LIN {X 0.018,Y -426.505,Z 505.911,A 0.000,B 0.000,C 90.000,E1 199.939} C_DIS
LIN {X 0.001,Y -422.220,Z 505.894,A 0.000,B 0.000,C 90.000,E1 196.913} C_DIS
LIN {X 0.056,Y -419.219,Z 505.881,A 0.000,B 0.000,C 90.000,E1 194.537} C_DIS
LIN {X -0.079,Y -416.405,Z 505.868,A 0.000,B 0.000,C 90.000,E1 192.175} C_DIS
LIN {X -0.186,Y -414.138,Z 505.856,A 0.000,B 0.000,C 90.000,E1 190.141} C_DIS
LIN {X 0.071,Y -411.990,Z 505.845,A 0.000,B 0.000,C 90.000,E1 188.049} C_DIS
LIN {X 0.180,Y -410.282,Z 505.835,A 0.000,B 0.000,C 90.000,E1 186.315} C_DIS
LIN {X 0.176,Y -407.524,Z 505.820,A 0.000,B 0.000,C 90.000,E1 183.555} C_DIS
LIN {X 0.039,Y -405.409,Z 505.805,A 0.000,B 0.000,C 90.000,E1 180.802} C_DIS
LIN {X -0.121,Y -404.165,Z 505.793,A 0.000,B 0.000,C 90.000,E1 178.740} C_DIS
LIN {X -0.033,Y -402.565,Z 505.770,A 0.000,B 0.000,C 90.000,E1 174.546} C_DIS
LIN {X 0.172,Y -402.279,Z 505.752,A 0.000,B 0.000,C 90.000,E1 171.376} C_DIS
LIN {X 0.214,Y -402.491,Z 505.739,A 0.000,B 0.000,C 90.000,E1 168.926} C_DIS
LIN {X -0.118,Y -402.858,Z 505.729,A 0.000,B 0.000,C 90.000,E1 167.229} C_DIS
LIN {X 0.210,Y -403.708,Z 505.714,A 0.000,B 0.000,C 90.000,E1 164.393} C_DIS
LIN {X 0.006,Y -405.079,Z 505.698,A 0.000,B 0.000,C 90.000,E1 161.638} C_DIS
LIN {X -0.119,Y -406.382,Z 505.686,A 0.000,B 0.000,C 90.000,E1 159.571} C_DIS
LIN {X 0.038,Y -409.257,Z 505.665,A 0.000,B 0.000,C 90.000,E1 155.741} C_DIS
LIN {X -0.103,Y -411.046,Z 505.654,A 0.000,B 0.000,C 90.000,E1 153.691} C_DIS
LIN {X -0.125,Y -412.516,Z 505.644,A 0.000,B 0.000,C 90.000,E1 151.975} C_DIS
LIN {X -0.098,Y -413.912,Z 505.635,A 0.000,B 0.000,C 90.000,E1 150.255} C_DIS
LIN {X -0.039,Y -415.256,Z 505.625,A 0.000,B 0.000,C 90.000,E1 148.535} C_DIS
LIN {X -0.093,Y -416.520,Z 505.616,A 0.000,B 0.000,C 90.000,E1 146.834} C_DIS
LIN {X 0.055,Y -417.849,Z 505.604,A 0.000,B 0.000,C 90.000,E1 144.769} C_DIS
LIN {X 0.184,Y -418.995,Z 505.595,A 0.000,B 0.000,C 90.000,E1 143.050} C_DIS
LIN {X 0.008,Y -420.032,Z 505.585,A 0.000,B 0.000,C 90.000,E1 141.376} C_DIS
LIN {X 0.116,Y -420.969,Z 505.576,A 0.000,B 0.000,C 90.000,E1 139.666} C_DIS
LIN {X 0.124,Y -421.898,Z 505.565,A 0.000,B 0.000,C 90.000,E1 137.634} C_DIS
LIN {X 0.116,Y -422.218,Z 505.559,A 0.000,B 0.000,C 90.000,E1 136.620} C_DIS
LIN {X 0.203,Y -422.557,Z 505.550,A 0.000,B 0.000,C 90.000,E1 134.919} C_DIS
LIN {X -0.099,Y -422.626,Z 505.544,A 0.000,B 0.000,C 90.000,E1 133.947} C_DIS
LIN {X -0.198,Y -422.402,Z 505.537,A 0.000,B 0.000,C 90.000,E1 132.609} C_DIS
LIN {X -0.199,Y -421.973,Z 505.531,A 0.000,B 0.000,C 90.000,E1 131.595} C_DIS
LIN {X -0.003,Y -421.086,Z 505.523,A 0.000,B 0.000,C 90.000,E1 130.216} C_DIS
LIN {X 0.024,Y -420.265,Z 505.518,A 0.000,B 0.000,C 90.000,E1 129.197} C_DIS
LIN {X -0.139,Y -418.800,Z 505.508,A 0.000,B 0.000,C 90.000,E1 127.523} C_DIS
LIN {X 0.000,Y -417.194,Z 505.499,A 0.000,B 0.000,C 90.000,E1 125.804} C_DIS
LIN {X -0.124,Y -416.814,Z 505.497,A 0.000,B 0.000,C 90.000,E1 125.438} C_DIS
LIN {X -0.161,Y -416.824,Z 505.497,A 0.000,B 0.000,C 90.000,E1 125.438} C_DIS
LIN {X 0.103,Y -426.391,Z 505.476,A 0.000,B 0.000,C 90.000,E1 121.720} C_DIS
LIN {X 0.058,Y -430.444,Z 505.469,A 0.000,B 0.000,C 90.000,E1 120.384} C_DIS
LIN {X -0.155,Y -432.036,Z 505.465,A 0.000,B 0.000,C 90.000,E1 119.745} C_DIS
LIN {X -0.164,Y -441.367,Z 505.445,A 0.000,B 0.000,C 90.000,E1 116.104} C_DIS
LIN {X 0.152,Y -444.273,Z 505.439,A 0.000,B 0.000,C 90.000,E1 115.079} C_DIS
LIN {X 0.005,Y -445.126,Z 505.438,A 0.000,B 0.000,C 90.000,E1 114.771} C_DIS
LIN {X 0.113,Y -454.300,Z 505.416,A 0.000,B 0.000,C 90.000,E1 110.865} C_DIS
LIN {X -0.196,Y -456.967,Z 505.411,A 0.000,B 0.000,C 90.000,E1 109.939} C_DIS
LIN {X 0.042,Y -458.234,Z 505.407,A 0.000,B 0.000,C 90.000,E1 109.268} C_DIS
LIN {X 0.191,Y -460.170,Z 505.401,A 0.000,B 0.000,C 90.000,E1 108.236} C_DIS
LIN {X 0.164,Y -460.188,Z 505.401,A 0.000,B 0.000,C 90.000,E1 108.236} C_DIS
LIN {X -0.031,Y -477.013,Z 505.399,A 0.000,B 0.000,C 90.000,E1 107.819} C_DIS
LIN {X 0.118,Y -487.752,Z 505.397,A 0.000,B 0.000,C 90.000,E1 107.511} C_DIS
LIN {X 0.183,Y -501.865,Z 505.395,A 0.000,B 0.000,C 90.000,E1 107.094} C_DIS
LIN {X -0.084,Y -512.281,Z 505.393,A 0.000,B 0.000,C 90.000,E1 106.804} C_DIS
LIN {X 0.104,Y -522.750,Z 505.391,A 0.000,B 0.000,C 90.000,E1 106.441} C_DIS
LIN {X 0.115,Y -533.203,Z 505.389,A 0.000,B 0.000,C 90.000,E1 106.079} C_DIS
LIN {X -0.021,Y -539.788,Z 505.388,A 0.000,B 0.000,C 90.000,E1 105.843} C_DIS
LIN {X 0.026,Y -549.515,Z 505.386,A 0.000,B 0.000,C 90.000,E1 105.426} C_DIS
LIN {X -0.055,Y -556.133,Z 505.384,A 0.000,B 0.000,C 90.000,E1 105.134} C_DIS
LIN {X -0.214,Y -562.178,Z 505.382,A 0.000,B 0.000,C 90.000,E1 104.828} C_DIS
LIN {X 0.204,Y -568.361,Z 505.380,A 0.000,B 0.000,C 90.000,E1 104.426} C_DIS
LIN {X -0.021,Y -574.397,Z 505.378,A 0.000,B 0.000,C 90.000,E1 104.064} C_DIS
LIN {X 0.015,Y -580.246,Z 505.376,A 0.000,B 0.000,C 90.000,E1 103.647} C_DIS
LIN {X -0.165,Y -585.770,Z 505.373,A 0.000,B 0.000,C 90.000,E1 103.231} C_DIS
LIN {X -0.180,Y -591.131,Z 505.371,A 0.000,B 0.000,C 90.000,E1 102.771} C_DIS
LIN {X -0.036,Y -598.036,Z 505.367,A 0.000,B 0.000,C 90.000,E1 102.119} C_DIS
LIN {X -0.101,Y -605.453,Z 505.363,A 0.000,B 0.000,C 90.000,E1 101.366} C_DIS
LIN {X -0.084,Y -609.662,Z 505.361,A 0.000,B 0.000,C 90.000,E1 100.894} C_DIS
LIN {X -0.103,Y -613.896,Z 505.358,A 0.000,B 0.000,C 90.000,E1 100.423} C_DIS
LIN {X 0.123,Y -618.926,Z 505.355,A 0.000,B 0.000,C 90.000,E1 99.792} C_DIS
LIN {X 0.104,Y -623.916,Z 505.351,A 0.000,B 0.000,C 90.000,E1 99.151} C_DIS
LIN {X -0.027,Y -629.277,Z 505.347,A 0.000,B 0.000,C 90.000,E1 98.398} C_DIS
LIN {X -0.108,Y -634.217,Z 505.342,A 0.000,B 0.000,C 90.000,E1 97.644} C_DIS
LIN {X -0.145,Y -638.618,Z 505.338,A 0.000,B 0.000,C 90.000,E1 96.891} C_DIS
LIN {X -0.088,Y -641.983,Z 505.335,A 0.000,B 0.000,C 90.000,E1 96.258} C_DIS
LIN {X 0.000,Y -645.065,Z 505.331,A 0.000,B 0.000,C 90.000,E1 95.625} C_DIS
LIN {X -0.178,Y -649.744,Z 505.326,A 0.000,B 0.000,C 90.000,E1 94.645} C_DIS
LIN {X -0.141,Y -652.900,Z 505.322,A 0.000,B 0.000,C 90.000,E1 93.898} C_DIS
LIN {X 0.094,Y -654.803,Z 505.319,A 0.000,B 0.000,C 90.000,E1 93.383} C_DIS
LIN {X -0.274,Y -656.487,Z 505.316,A 0.000,B 0.000,C 90.000,E1 92.922} C_DIS
LIN {X -0.010,Y -657.988,Z 505.313,A 0.000,B 0.000,C 90.000,E1 92.407} C_DIS
LIN {X 0.105,Y -659.741,Z 505.309,A 0.000,B 0.000,C 90.000,E1 91.661} C_DIS
LIN {X -0.264,Y -660.700,Z 505.307,A 0.000,B 0.000,C 90.000,E1 91.203} C_DIS
LIN {X 0.037,Y -661.322,Z 505.304,A 0.000,B 0.000,C 90.000,E1 90.688} C_DIS
LIN {X -0.319,Y -661.735,Z 505.301,A 0.000,B 0.000,C 90.000,E1 90.229} C_DIS
LIN {X -0.009,Y -661.834,Z 505.298,A 0.000,B 0.000,C 90.000,E1 89.714} C_DIS
LIN {X 0.126,Y -661.721,Z 505.294,A 0.000,B 0.000,C 90.000,E1 88.969} C_DIS
LIN {X 0.255,Y -661.045,Z 505.290,A 0.000,B 0.000,C 90.000,E1 88.224} C_DIS
LIN {X -0.080,Y -660.385,Z 505.288,A 0.000,B 0.000,C 90.000,E1 87.764} C_DIS
LIN {X 0.032,Y -658.956,Z 505.284,A 0.000,B 0.000,C 90.000,E1 87.020} C_DIS
LIN {X -0.305,Y -657.826,Z 505.281,A 0.000,B 0.000,C 90.000,E1 86.560} C_DIS
LIN {X -0.032,Y -656.465,Z 505.278,A 0.000,B 0.000,C 90.000,E1 86.045} C_DIS
LIN {X 0.275,Y -654.873,Z 505.275,A 0.000,B 0.000,C 90.000,E1 85.527} C_DIS
LIN {X -0.287,Y -652.156,Z 505.271,A 0.000,B 0.000,C 90.000,E1 84.837} C_DIS
LIN {X -0.004,Y -650.150,Z 505.268,A 0.000,B 0.000,C 90.000,E1 84.318} C_DIS
LIN {X 0.036,Y -646.773,Z 505.264,A 0.000,B 0.000,C 90.000,E1 83.571} C_DIS
LIN {X 0.279,Y -644.240,Z 505.262,A 0.000,B 0.000,C 90.000,E1 83.053} C_DIS
LIN {X -0.180,Y -640.958,Z 505.258,A 0.000,B 0.000,C 90.000,E1 82.470} C_DIS
LIN {X -0.058,Y -636.731,Z 505.254,A 0.000,B 0.000,C 90.000,E1 81.724} C_DIS
LIN {X -0.022,Y -630.363,Z 505.249,A 0.000,B 0.000,C 90.000,E1 80.735} C_DIS
LIN {X -0.110,Y -624.978,Z 505.244,A 0.000,B 0.000,C 90.000,E1 79.982} C_DIS
LIN {X 0.086,Y -619.367,Z 505.240,A 0.000,B 0.000,C 90.000,E1 79.218} C_DIS
LIN {X 0.134,Y -614.176,Z 505.237,A 0.000,B 0.000,C 90.000,E1 78.578} C_DIS
LIN {X 0.062,Y -608.507,Z 505.233,A 0.000,B 0.000,C 90.000,E1 77.937} C_DIS
LIN {X 0.169,Y -603.608,Z 505.230,A 0.000,B 0.000,C 90.000,E1 77.409} C_DIS
LIN {X -0.064,Y -598.510,Z 505.227,A 0.000,B 0.000,C 90.000,E1 76.937} C_DIS
LIN {X -0.120,Y -593.055,Z 505.225,A 0.000,B 0.000,C 90.000,E1 76.464} C_DIS
LIN {X 0.014,Y -587.480,Z 505.222,A 0.000,B 0.000,C 90.000,E1 75.992} C_DIS
LIN {X 0.273,Y -581.520,Z 505.220,A 0.000,B 0.000,C 90.000,E1 75.519} C_DIS
LIN {X -0.186,Y -575.580,Z 505.218,A 0.000,B 0.000,C 90.000,E1 75.172} C_DIS
LIN {X -0.012,Y -570.706,Z 505.216,A 0.000,B 0.000,C 90.000,E1 74.866} C_DIS
LIN {X -0.110,Y -563.793,Z 505.214,A 0.000,B 0.000,C 90.000,E1 74.519} C_DIS
LIN {X -0.172,Y -558.480,Z 505.213,A 0.000,B 0.000,C 90.000,E1 74.283} C_DIS
LIN {X 0.162,Y -553.060,Z 505.211,A 0.000,B 0.000,C 90.000,E1 74.031} C_DIS
LIN {X 0.016,Y -545.580,Z 505.210,A 0.000,B 0.000,C 90.000,E1 73.795} C_DIS
LIN {X 0.160,Y -539.833,Z 505.209,A 0.000,B 0.000,C 90.000,E1 73.614} C_DIS
LIN {X 0.030,Y -532.141,Z 505.208,A 0.000,B 0.000,C 90.000,E1 73.449} C_DIS
LIN {X -0.123,Y -523.817,Z 505.207,A 0.000,B 0.000,C 90.000,E1 73.323} C_DIS
LIN {X -0.043,Y -511.657,Z 505.206,A 0.000,B 0.000,C 90.000,E1 73.142} C_DIS
LIN {X 0.061,Y -500.841,Z 505.206,A 0.000,B 0.000,C 90.000,E1 73.015} C_DIS
LIN {X 0.175,Y -495.888,Z 505.206,A 0.000,B 0.000,C 90.000,E1 72.960} C_DIS
LIN {X -0.166,Y -488.331,Z 505.205,A 0.000,B 0.000,C 90.000,E1 72.960} C_DIS
LIN {X 0.119,Y -478.178,Z 505.205,A 0.000,B 0.000,C 90.000,E1 72.851} C_DIS
LIN {X -0.010,Y -474.985,Z 505.205,A 0.000,B 0.000,C 90.000,E1 72.851} C_DIS
LIN {X -0.042,Y -474.946,Z 505.205,A 0.000,B 0.000,C 90.000,E1 72.851} C_DIS
LIN {X 0.221,Y -474.159,Z 505.201,A 0.000,B 0.000,C 90.000,E1 72.054} C_DIS
LIN {X 0.088,Y -465.644,Z 505.173,A 0.000,B 0.000,C 90.000,E1 67.050} C_DIS
LIN {X -0.033,Y -456.637,Z 505.148,A 0.000,B 0.000,C 90.000,E1 62.615} C_DIS
LIN {X -0.034,Y -455.594,Z 505.144,A 0.000,B 0.000,C 90.000,E1 61.975} C_DIS
LIN {X 0.150,Y -452.503,Z 505.137,A 0.000,B 0.000,C 90.000,E1 60.667} C_DIS
LIN {X -0.182,Y -448.840,Z 505.128,A 0.000,B 0.000,C 90.000,E1 59.076} C_DIS
LIN {X -0.221,Y -448.858,Z 505.128,A 0.000,B 0.000,C 90.000,E1 59.076} C_DIS
LIN {X 0.196,Y -453.401,Z 505.122,A 0.000,B 0.000,C 90.000,E1 57.916} C_DIS
LIN {X 0.110,Y -457.127,Z 505.117,A 0.000,B 0.000,C 90.000,E1 56.962} C_DIS
LIN {X -0.044,Y -458.885,Z 505.114,A 0.000,B 0.000,C 90.000,E1 56.501} C_DIS
LIN {X -0.200,Y -461.027,Z 505.110,A 0.000,B 0.000,C 90.000,E1 55.881} C_DIS
LIN {X 0.048,Y -463.771,Z 505.105,A 0.000,B 0.000,C 90.000,E1 54.895} C_DIS
LIN {X -0.072,Y -465.454,Z 505.102,A 0.000,B 0.000,C 90.000,E1 54.276} C_DIS
LIN {X -0.145,Y -467.569,Z 505.096,A 0.000,B 0.000,C 90.000,E1 53.336} C_DIS
LIN {X 0.042,Y -468.814,Z 505.093,A 0.000,B 0.000,C 90.000,E1 52.683} C_DIS
LIN {X 0.013,Y -470.423,Z 505.088,A 0.000,B 0.000,C 90.000,E1 51.743} C_DIS
LIN {X -0.148,Y -472.508,Z 505.079,A 0.000,B 0.000,C 90.000,E1 50.194} C_DIS
LIN {X -0.059,Y -473.786,Z 505.072,A 0.000,B 0.000,C 90.000,E1 48.933} C_DIS
LIN {X -0.093,Y -474.575,Z 505.067,A 0.000,B 0.000,C 90.000,E1 48.000} C_DIS
LIN {X -0.115,Y -475.209,Z 505.061,A 0.000,B 0.000,C 90.000,E1 47.067} C_DIS
LIN {X -0.132,Y -475.735,Z 505.056,A 0.000,B 0.000,C 90.000,E1 46.134} C_DIS
LIN {X 0.187,Y -476.122,Z 505.051,A 0.000,B 0.000,C 90.000,E1 45.162} C_DIS
LIN {X -0.055,Y -476.457,Z 505.044,A 0.000,B 0.000,C 90.000,E1 43.947} C_DIS
LIN {X 0.050,Y -476.486,Z 505.037,A 0.000,B 0.000,C 90.000,E1 42.690} C_DIS
LIN {X 0.152,Y -476.221,Z 505.030,A 0.000,B 0.000,C 90.000,E1 41.434} C_DIS
LIN {X -0.171,Y -475.911,Z 505.025,A 0.000,B 0.000,C 90.000,E1 40.539} C_DIS
LIN {X 0.059,Y -475.261,Z 505.017,A 0.000,B 0.000,C 90.000,E1 38.955} C_DIS
LIN {X 0.133,Y -474.287,Z 505.006,A 0.000,B 0.000,C 90.000,E1 37.076} C_DIS
LIN {X -0.098,Y -473.158,Z 504.996,A 0.000,B 0.000,C 90.000,E1 35.231} C_DIS
LIN {X -0.016,Y -472.070,Z 504.987,A 0.000,B 0.000,C 90.000,E1 33.658} C_DIS
LIN {X -0.011,Y -470.371,Z 504.975,A 0.000,B 0.000,C 90.000,E1 31.465} C_DIS
LIN {X -0.075,Y -468.725,Z 504.964,A 0.000,B 0.000,C 90.000,E1 29.589} C_DIS
LIN {X -0.226,Y -467.068,Z 504.954,A 0.000,B 0.000,C 90.000,E1 27.719} C_DIS
LIN {X 0.012,Y -465.525,Z 504.943,A 0.000,B 0.000,C 90.000,E1 25.796} C_DIS
LIN {X 0.013,Y -464.076,Z 504.933,A 0.000,B 0.000,C 90.000,E1 23.898} C_DIS
LIN {X -0.143,Y -463.094,Z 504.924,A 0.000,B 0.000,C 90.000,E1 22.333} C_DIS
LIN {X -0.138,Y -462.053,Z 504.913,A 0.000,B 0.000,C 90.000,E1 20.429} C_DIS
LIN {X 0.122,Y -461.156,Z 504.903,A 0.000,B 0.000,C 90.000,E1 18.489} C_DIS
LIN {X -0.090,Y -460.199,Z 504.889,A 0.000,B 0.000,C 90.000,E1 15.969} C_DIS
LIN {X -0.025,Y -459.576,Z 504.875,A 0.000,B 0.000,C 90.000,E1 13.411} C_DIS
LIN {X -0.068,Y -459.439,Z 504.859,A 0.000,B 0.000,C 90.000,E1 10.546} C_DIS
LIN {X 0.229,Y -459.695,Z 504.846,A 0.000,B 0.000,C 90.000,E1 8.276} C_DIS
LIN {X -0.113,Y -460.288,Z 504.834,A 0.000,B 0.000,C 90.000,E1 6.087} C_DIS
LIN {X 0.026,Y -461.345,Z 504.821,A 0.000,B 0.000,C 90.000,E1 3.841} C_DIS
LIN {X -0.104,Y -462.522,Z 504.811,A 0.000,B 0.000,C 90.000,E1 1.949} C_DIS
LIN {X 0.000,Y -463.977,Z 504.800,A 0.000,B 0.000,C 90.000,E1 360.000} C_DIS
LIN {X -0.123,Y -466.352,Z 504.787,A 0.000,B 0.000,C 90.000,E1 357.593} C_DIS
LIN {X -0.128,Y -467.758,Z 504.780,A 0.000,B 0.000,C 90.000,E1 356.331} C_DIS
LIN {X -0.046,Y -470.034,Z 504.769,A 0.000,B 0.000,C 90.000,E1 354.432} C_DIS
LIN {X 0.038,Y -471.673,Z 504.762,A 0.000,B 0.000,C 90.000,E1 353.166} C_DIS
LIN {X 0.028,Y -473.689,Z 504.753,A 0.000,B 0.000,C 90.000,E1 351.602} C_DIS
LIN {X -0.109,Y -477.718,Z 504.738,A 0.000,B 0.000,C 90.000,E1 348.814} C_DIS
LIN {X 0.182,Y -482.461,Z 504.722,A 0.000,B 0.000,C 90.000,E1 345.992} C_DIS
LIN {X -0.059,Y -486.669,Z 504.710,A 0.000,B 0.000,C 90.000,E1 343.866} C_DIS
LIN {X 0.069,Y -491.080,Z 504.698,A 0.000,B 0.000,C 90.000,E1 341.710} C_DIS
LIN {X 0.038,Y -493.709,Z 504.692,A 0.000,B 0.000,C 90.000,E1 340.496} C_DIS
LIN {X 0.219,Y -496.330,Z 504.685,A 0.000,B 0.000,C 90.000,E1 339.263} C_DIS
LIN {X -0.198,Y -498.964,Z 504.678,A 0.000,B 0.000,C 90.000,E1 338.103} C_DIS
LIN {X 0.135,Y -502.099,Z 504.670,A 0.000,B 0.000,C 90.000,E1 336.561} C_DIS
LIN {X 0.186,Y -504.564,Z 504.663,A 0.000,B 0.000,C 90.000,E1 335.357} C_DIS
LIN {X -0.003,Y -508.099,Z 504.653,A 0.000,B 0.000,C 90.000,E1 333.589} C_DIS
LIN {X -0.108,Y -511.728,Z 504.643,A 0.000,B 0.000,C 90.000,E1 331.820} C_DIS
LIN {X -0.117,Y -515.345,Z 504.634,A 0.000,B 0.000,C 90.000,E1 330.049} C_DIS
LIN {X 0.281,Y -518.532,Z 504.625,A 0.000,B 0.000,C 90.000,E1 328.535} C_DIS
LIN {X 0.174,Y -522.910,Z 504.614,A 0.000,B 0.000,C 90.000,E1 326.501} C_DIS
LIN {X 0.029,Y -527.428,Z 504.603,A 0.000,B 0.000,C 90.000,E1 324.482} C_DIS
LIN {X -0.106,Y -531.268,Z 504.593,A 0.000,B 0.000,C 90.000,E1 322.763} C_DIS
LIN {X -0.159,Y -534.444,Z 504.585,A 0.000,B 0.000,C 90.000,E1 321.331} C_DIS
LIN {X -0.241,Y -537.576,Z 504.577,A 0.000,B 0.000,C 90.000,E1 319.908} C_DIS
LIN {X 0.103,Y -541.341,Z 504.568,A 0.000,B 0.000,C 90.000,E1 318.162} C_DIS
LIN {X 0.124,Y -545.103,Z 504.558,A 0.000,B 0.000,C 90.000,E1 316.458} C_DIS
LIN {X 0.209,Y -548.704,Z 504.549,A 0.000,B 0.000,C 90.000,E1 314.757} C_DIS
LIN {X -0.052,Y -551.588,Z 504.541,A 0.000,B 0.000,C 90.000,E1 313.380} C_DIS
LIN {X 0.190,Y -555.091,Z 504.532,A 0.000,B 0.000,C 90.000,E1 311.676} C_DIS
LIN {X 0.062,Y -558.036,Z 504.524,A 0.000,B 0.000,C 90.000,E1 310.297} C_DIS
LIN {X 0.148,Y -561.549,Z 504.515,A 0.000,B 0.000,C 90.000,E1 308.624} C_DIS
LIN {X -0.022,Y -565.611,Z 504.504,A 0.000,B 0.000,C 90.000,E1 306.710} C_DIS
LIN {X -0.326,Y -569.663,Z 504.493,A 0.000,B 0.000,C 90.000,E1 304.818} C_DIS
LIN {X -0.191,Y -573.145,Z 504.484,A 0.000,B 0.000,C 90.000,E1 303.166} C_DIS
LIN {X -0.128,Y -575.988,Z 504.477,A 0.000,B 0.000,C 90.000,E1 301.799} C_DIS
LIN {X -0.169,Y -578.181,Z 504.471,A 0.000,B 0.000,C 90.000,E1 300.718} C_DIS
LIN {X 0.173,Y -580.786,Z 504.463,A 0.000,B 0.000,C 90.000,E1 299.333} C_DIS
LIN {X -0.231,Y -583.361,Z 504.456,A 0.000,B 0.000,C 90.000,E1 298.025} C_DIS
LIN {X -0.080,Y -585.405,Z 504.448,A 0.000,B 0.000,C 90.000,E1 296.668} C_DIS
LIN {X -0.156,Y -587.042,Z 504.441,A 0.000,B 0.000,C 90.000,E1 295.335} C_DIS
LIN {X 0.026,Y -587.805,Z 504.436,A 0.000,B 0.000,C 90.000,E1 294.515} C_DIS
LIN {X 0.176,Y -588.749,Z 504.427,A 0.000,B 0.000,C 90.000,E1 292.898} C_DIS
LIN {X 0.014,Y -589.864,Z 504.417,A 0.000,B 0.000,C 90.000,E1 291.046} C_DIS
LIN {X -0.012,Y -590.652,Z 504.408,A 0.000,B 0.000,C 90.000,E1 289.450} C_DIS
LIN {X 0.216,Y -590.968,Z 504.402,A 0.000,B 0.000,C 90.000,E1 288.362} C_DIS
LIN {X 0.136,Y -591.213,Z 504.395,A 0.000,B 0.000,C 90.000,E1 287.040} C_DIS
LIN {X 0.200,Y -591.371,Z 504.389,A 0.000,B 0.000,C 90.000,E1 285.969} C_DIS
LIN {X -0.036,Y -591.454,Z 504.382,A 0.000,B 0.000,C 90.000,E1 284.662} C_DIS
LIN {X -0.010,Y -591.469,Z 504.373,A 0.000,B 0.000,C 90.000,E1 283.063} C_DIS
LIN {X 0.145,Y -591.396,Z 504.362,A 0.000,B 0.000,C 90.000,E1 281.186} C_DIS
LIN {X -0.092,Y -591.179,Z 504.353,A 0.000,B 0.000,C 90.000,E1 279.613} C_DIS
LIN {X -0.023,Y -590.906,Z 504.346,A 0.000,B 0.000,C 90.000,E1 278.276} C_DIS
LIN {X 0.138,Y -590.415,Z 504.337,A 0.000,B 0.000,C 90.000,E1 276.663} C_DIS
LIN {X -0.146,Y -589.943,Z 504.331,A 0.000,B 0.000,C 90.000,E1 275.625} C_DIS
LIN {X -0.008,Y -588.999,Z 504.322,A 0.000,B 0.000,C 90.000,E1 274.012} C_DIS
LIN {X -0.172,Y -587.921,Z 504.315,A 0.000,B 0.000,C 90.000,E1 272.694} C_DIS
LIN {X 0.236,Y -586.563,Z 504.307,A 0.000,B 0.000,C 90.000,E1 271.318} C_DIS
LIN {X -0.171,Y -585.335,Z 504.302,A 0.000,B 0.000,C 90.000,E1 270.286} C_DIS
LIN {X -0.224,Y -583.438,Z 504.293,A 0.000,B 0.000,C 90.000,E1 268.682} C_DIS
LIN {X 0.273,Y -581.327,Z 504.284,A 0.000,B 0.000,C 90.000,E1 267.020} C_DIS
LIN {X 0.015,Y -579.543,Z 504.276,A 0.000,B 0.000,C 90.000,E1 265.698} C_DIS
LIN {X -0.266,Y -577.635,Z 504.269,A 0.000,B 0.000,C 90.000,E1 264.375} C_DIS
LIN {X 0.185,Y -575.024,Z 504.260,A 0.000,B 0.000,C 90.000,E1 262.704} C_DIS
LIN {X 0.079,Y -572.312,Z 504.251,A 0.000,B 0.000,C 90.000,E1 261.084} C_DIS
LIN {X 0.008,Y -569.624,Z 504.241,A 0.000,B 0.000,C 90.000,E1 259.454} C_DIS
LIN {X -0.186,Y -567.135,Z 504.234,A 0.000,B 0.000,C 90.000,E1 258.105} C_DIS
LIN {X -0.038,Y -565.167,Z 504.228,A 0.000,B 0.000,C 90.000,E1 256.992} C_DIS
LIN {X 0.075,Y -563.100,Z 504.222,A 0.000,B 0.000,C 90.000,E1 255.880} C_DIS
LIN {X -0.108,Y -560.304,Z 504.214,A 0.000,B 0.000,C 90.000,E1 254.519} C_DIS
LIN {X -0.186,Y -557.330,Z 504.206,A 0.000,B 0.000,C 90.000,E1 253.142} C_DIS
LIN {X -0.035,Y -553.406,Z 504.197,A 0.000,B 0.000,C 90.000,E1 251.456} C_DIS
LIN {X 0.098,Y -551.385,Z 504.192,A 0.000,B 0.000,C 90.000,E1 250.604} C_DIS
LIN {X 0.033,Y -547.744,Z 504.185,A 0.000,B 0.000,C 90.000,E1 249.209} C_DIS
LIN {X 0.091,Y -544.010,Z 504.177,A 0.000,B 0.000,C 90.000,E1 247.794} C_DIS
LIN {X 0.287,Y -540.067,Z 504.169,A 0.000,B 0.000,C 90.000,E1 246.357} C_DIS
LIN {X 0.196,Y -536.721,Z 504.163,A 0.000,B 0.000,C 90.000,E1 245.229} C_DIS
LIN {X 0.195,Y -531.571,Z 504.153,A 0.000,B 0.000,C 90.000,E1 243.512} C_DIS
LIN {X -0.147,Y -526.240,Z 504.143,A 0.000,B 0.000,C 90.000,E1 241.820} C_DIS
LIN {X -0.209,Y -519.944,Z 504.132,A 0.000,B 0.000,C 90.000,E1 239.793} C_DIS
LIN {X -0.197,Y -515.403,Z 504.124,A 0.000,B 0.000,C 90.000,E1 238.329} C_DIS
LIN {X -0.002,Y -510.726,Z 504.116,A 0.000,B 0.000,C 90.000,E1 236.834} C_DIS
LIN {X -0.007,Y -504.940,Z 504.106,A 0.000,B 0.000,C 90.000,E1 235.055} C_DIS
LIN {X 0.029,Y -499.215,Z 504.096,A 0.000,B 0.000,C 90.000,E1 233.256} C_DIS
LIN {X -0.195,Y -492.849,Z 504.084,A 0.000,B 0.000,C 90.000,E1 231.170} C_DIS
LIN {X 0.194,Y -487.664,Z 504.074,A 0.000,B 0.000,C 90.000,E1 229.299} C_DIS
LIN {X 0.227,Y -481.919,Z 504.062,A 0.000,B 0.000,C 90.000,E1 227.148} C_DIS
LIN {X -0.029,Y -476.996,Z 504.052,A 0.000,B 0.000,C 90.000,E1 225.324} C_DIS
LIN {X 0.030,Y -471.503,Z 504.040,A 0.000,B 0.000,C 90.000,E1 223.137} C_DIS
LIN {X -0.007,Y -466.207,Z 504.027,A 0.000,B 0.000,C 90.000,E1 220.943} C_DIS
LIN {X -0.177,Y -461.262,Z 504.015,A 0.000,B 0.000,C 90.000,E1 218.749} C_DIS
LIN {X 0.206,Y -457.145,Z 504.005,A 0.000,B 0.000,C 90.000,E1 216.790} C_DIS
LIN {X 0.046,Y -452.546,Z 503.992,A 0.000,B 0.000,C 90.000,E1 214.565} C_DIS
LIN {X -0.157,Y -447.570,Z 503.978,A 0.000,B 0.000,C 90.000,E1 212.005} C_DIS
LIN {X -0.128,Y -443.975,Z 503.967,A 0.000,B 0.000,C 90.000,E1 210.050} C_DIS
LIN {X 0.229,Y -439.275,Z 503.952,A 0.000,B 0.000,C 90.000,E1 207.385} C_DIS
LIN {X -0.192,Y -435.760,Z 503.941,A 0.000,B 0.000,C 90.000,E1 205.463} C_DIS
LIN {X -0.087,Y -432.341,Z 503.930,A 0.000,B 0.000,C 90.000,E1 203.462} C_DIS
LIN {X -0.065,Y -429.010,Z 503.919,A 0.000,B 0.000,C 90.000,E1 201.461} C_DIS
LIN {X 0.160,Y -426.426,Z 503.910,A 0.000,B 0.000,C 90.000,E1 199.758} C_DIS
LIN {X -0.044,Y -422.596,Z 503.895,A 0.000,B 0.000,C 90.000,E1 197.094} C_DIS
LIN {X 0.024,Y -419.551,Z 503.882,A 0.000,B 0.000,C 90.000,E1 194.717} C_DIS
LIN {X -0.098,Y -416.705,Z 503.869,A 0.000,B 0.000,C 90.000,E1 192.355} C_DIS
LIN {X -0.072,Y -414.060,Z 503.855,A 0.000,B 0.000,C 90.000,E1 189.962} C_DIS
LIN {X 0.174,Y -411.896,Z 503.844,A 0.000,B 0.000,C 90.000,E1 187.871} C_DIS
LIN {X -0.179,Y -410.198,Z 503.834,A 0.000,B 0.000,C 90.000,E1 186.201} C_DIS
LIN {X -0.170,Y -408.124,Z 503.823,A 0.000,B 0.000,C 90.000,E1 184.131} C_DIS
LIN {X 0.115,Y -405.631,Z 503.806,A 0.000,B 0.000,C 90.000,E1 180.974} C_DIS
LIN {X -0.038,Y -404.364,Z 503.794,A 0.000,B 0.000,C 90.000,E1 178.912} C_DIS
LIN {X 0.023,Y -402.698,Z 503.771,A 0.000,B 0.000,C 90.000,E1 174.723} C_DIS
LIN {X -0.116,Y -402.362,Z 503.755,A 0.000,B 0.000,C 90.000,E1 171.951} C_DIS
LIN {X -0.137,Y -402.522,Z 503.742,A 0.000,B 0.000,C 90.000,E1 169.511} C_DIS
LIN {X -0.001,Y -403.093,Z 503.726,A 0.000,B 0.000,C 90.000,E1 166.700} C_DIS
LIN {X -0.059,Y -404.083,Z 503.711,A 0.000,B 0.000,C 90.000,E1 163.921} C_DIS
LIN {X -0.023,Y -405.755,Z 503.693,A 0.000,B 0.000,C 90.000,E1 160.786} C_DIS
LIN {X 0.137,Y -406.872,Z 503.684,A 0.000,B 0.000,C 90.000,E1 159.028} C_DIS
LIN {X 0.077,Y -408.713,Z 503.670,A 0.000,B 0.000,C 90.000,E1 156.613} C_DIS
LIN {X -0.164,Y -410.206,Z 503.661,A 0.000,B 0.000,C 90.000,E1 154.921} C_DIS
LIN {X -0.019,Y -411.753,Z 503.651,A 0.000,B 0.000,C 90.000,E1 153.179} C_DIS
LIN {X 0.165,Y -413.228,Z 503.641,A 0.000,B 0.000,C 90.000,E1 151.435} C_DIS
LIN {X 0.067,Y -414.353,Z 503.634,A 0.000,B 0.000,C 90.000,E1 150.078} C_DIS
LIN {X -0.064,Y -416.005,Z 503.622,A 0.000,B 0.000,C 90.000,E1 148.043} C_DIS
LIN {X -0.096,Y -417.259,Z 503.613,A 0.000,B 0.000,C 90.000,E1 146.342} C_DIS
LIN {X 0.123,Y -418.418,Z 503.604,A 0.000,B 0.000,C 90.000,E1 144.609} C_DIS
LIN {X 0.017,Y -419.571,Z 503.594,A 0.000,B 0.000,C 90.000,E1 142.924} C_DIS
LIN {X -0.154,Y -420.683,Z 503.585,A 0.000,B 0.000,C 90.000,E1 141.251} C_DIS
LIN {X -0.247,Y -421.474,Z 503.577,A 0.000,B 0.000,C 90.000,E1 139.908} C_DIS
LIN {X 0.159,Y -422.345,Z 503.568,A 0.000,B 0.000,C 90.000,E1 138.162} C_DIS
LIN {X 0.058,Y -422.903,Z 503.560,A 0.000,B 0.000,C 90.000,E1 136.824} C_DIS
LIN {X -0.034,Y -423.206,Z 503.553,A 0.000,B 0.000,C 90.000,E1 135.486} C_DIS
LIN {X -0.032,Y -423.390,Z 503.547,A 0.000,B 0.000,C 90.000,E1 134.474} C_DIS
LIN {X 0.074,Y -423.436,Z 503.543,A 0.000,B 0.000,C 90.000,E1 133.785} C_DIS
LIN {X 0.087,Y -423.289,Z 503.538,A 0.000,B 0.000,C 90.000,E1 132.771} C_DIS
LIN {X -0.008,Y -422.696,Z 503.530,A 0.000,B 0.000,C 90.000,E1 131.434} C_DIS
LIN {X -0.074,Y -421.787,Z 503.523,A 0.000,B 0.000,C 90.000,E1 130.092} C_DIS
LIN {X -0.033,Y -420.930,Z 503.517,A 0.000,B 0.000,C 90.000,E1 129.072} C_DIS
LIN {X 0.076,Y -419.379,Z 503.508,A 0.000,B 0.000,C 90.000,E1 127.363} C_DIS
LIN {X -0.023,Y -417.705,Z 503.498,A 0.000,B 0.000,C 90.000,E1 125.678} C_DIS
LIN {X 0.129,Y -417.221,Z 503.496,A 0.000,B 0.000,C 90.000,E1 125.231} C_DIS
LIN {X 0.091,Y -417.222,Z 503.496,A 0.000,B 0.000,C 90.000,E1 125.231} C_DIS
LIN {X 0.106,Y -426.762,Z 503.476,A 0.000,B 0.000,C 90.000,E1 121.592} C_DIS
LIN {X 0.068,Y -430.820,Z 503.468,A 0.000,B 0.000,C 90.000,E1 120.256} C_DIS
LIN {X 0.028,Y -440.784,Z 503.446,A 0.000,B 0.000,C 90.000,E1 116.283} C_DIS
LIN {X -0.002,Y -444.651,Z 503.439,A 0.000,B 0.000,C 90.000,E1 114.975} C_DIS
LIN {X 0.159,Y -454.628,Z 503.415,A 0.000,B 0.000,C 90.000,E1 110.737} C_DIS
LIN {X -0.149,Y -457.289,Z 503.410,A 0.000,B 0.000,C 90.000,E1 109.812} C_DIS
LIN {X -0.026,Y -460.957,Z 503.399,A 0.000,B 0.000,C 90.000,E1 107.873} C_DIS
LIN {X -0.070,Y -461.099,Z 503.399,A 0.000,B 0.000,C 90.000,E1 107.873} C_DIS
LIN {X -0.217,Y -474.105,Z 503.398,A 0.000,B 0.000,C 90.000,E1 107.583} C_DIS
LIN {X 0.094,Y -484.730,Z 503.396,A 0.000,B 0.000,C 90.000,E1 107.275} C_DIS
LIN {X -0.120,Y -498.663,Z 503.394,A 0.000,B 0.000,C 90.000,E1 106.913} C_DIS
LIN {X -0.084,Y -512.752,Z 503.392,A 0.000,B 0.000,C 90.000,E1 106.496} C_DIS
LIN {X 0.183,Y -523.110,Z 503.390,A 0.000,B 0.000,C 90.000,E1 106.134} C_DIS
LIN {X 0.142,Y -533.576,Z 503.388,A 0.000,B 0.000,C 90.000,E1 105.788} C_DIS
LIN {X 0.049,Y -540.199,Z 503.386,A 0.000,B 0.000,C 90.000,E1 105.552} C_DIS
LIN {X 0.087,Y -550.147,Z 503.384,A 0.000,B 0.000,C 90.000,E1 105.134} C_DIS
LIN {X 0.150,Y -556.666,Z 503.383,A 0.000,B 0.000,C 90.000,E1 104.828} C_DIS
LIN {X -0.292,Y -559.837,Z 503.382,A 0.000,B 0.000,C 90.000,E1 104.717} C_DIS
LIN {X -0.076,Y -566.062,Z 503.380,A 0.000,B 0.000,C 90.000,E1 104.356} C_DIS
LIN {X -0.048,Y -569.090,Z 503.379,A 0.000,B 0.000,C 90.000,E1 104.175} C_DIS
LIN {X 0.042,Y -575.036,Z 503.377,A 0.000,B 0.000,C 90.000,E1 103.772} C_DIS
LIN {X 0.004,Y -580.484,Z 503.375,A 0.000,B 0.000,C 90.000,E1 103.411} C_DIS
LIN {X -0.150,Y -587.398,Z 503.372,A 0.000,B 0.000,C 90.000,E1 102.883} C_DIS
LIN {X -0.167,Y -591.560,Z 503.370,A 0.000,B 0.000,C 90.000,E1 102.535} C_DIS
LIN {X -0.147,Y -594.136,Z 503.368,A 0.000,B 0.000,C 90.000,E1 102.299} C_DIS
LIN {X -0.258,Y -596.456,Z 503.367,A 0.000,B 0.000,C 90.000,E1 102.119} C_DIS
LIN {X 0.201,Y -600.085,Z 503.365,A 0.000,B 0.000,C 90.000,E1 101.715} C_DIS
LIN {X -0.043,Y -603.906,Z 503.363,A 0.000,B 0.000,C 90.000,E1 101.366} C_DIS
LIN {X 0.075,Y -608.343,Z 503.361,A 0.000,B 0.000,C 90.000,E1 100.894} C_DIS
LIN {X 0.167,Y -613.131,Z 503.358,A 0.000,B 0.000,C 90.000,E1 100.366} C_DIS
LIN {X -0.069,Y -619.675,Z 503.353,A 0.000,B 0.000,C 90.000,E1 99.613} C_DIS
LIN {X -0.084,Y -624.747,Z 503.350,A 0.000,B 0.000,C 90.000,E1 98.973} C_DIS
LIN {X 0.261,Y -630.912,Z 503.345,A 0.000,B 0.000,C 90.000,E1 98.049} C_DIS
LIN {X -0.235,Y -634.225,Z 503.342,A 0.000,B 0.000,C 90.000,E1 97.587} C_DIS
LIN {X -0.271,Y -638.689,Z 503.338,A 0.000,B 0.000,C 90.000,E1 96.834} C_DIS
LIN {X -0.213,Y -642.067,Z 503.334,A 0.000,B 0.000,C 90.000,E1 96.201} C_DIS
LIN {X -0.124,Y -645.163,Z 503.331,A 0.000,B 0.000,C 90.000,E1 95.568} C_DIS
LIN {X -0.297,Y -649.873,Z 503.325,A 0.000,B 0.000,C 90.000,E1 94.588} C_DIS
LIN {X -0.258,Y -653.046,Z 503.321,A 0.000,B 0.000,C 90.000,E1 93.841} C_DIS
LIN {X -0.023,Y -654.939,Z 503.319,A 0.000,B 0.000,C 90.000,E1 93.326} C_DIS
LIN {X 0.069,Y -657.375,Z 503.314,A 0.000,B 0.000,C 90.000,E1 92.579} C_DIS
LIN {X -0.316,Y -658.702,Z 503.312,A 0.000,B 0.000,C 90.000,E1 92.121} C_DIS
LIN {X 0.157,Y -659.313,Z 503.310,A 0.000,B 0.000,C 90.000,E1 91.835} C_DIS
LIN {X -0.194,Y -660.289,Z 503.308,A 0.000,B 0.000,C 90.000,E1 91.375} C_DIS
LIN {X 0.102,Y -660.997,Z 503.305,A 0.000,B 0.000,C 90.000,E1 90.859} C_DIS
LIN {X -0.255,Y -661.489,Z 503.302,A 0.000,B 0.000,C 90.000,E1 90.401} C_DIS
LIN {X 0.230,Y -661.701,Z 503.301,A 0.000,B 0.000,C 90.000,E1 90.115} C_DIS
LIN {X -0.299,Y -661.683,Z 503.297,A 0.000,B 0.000,C 90.000,E1 89.427} C_DIS
LIN {X 0.011,Y -661.508,Z 503.294,A 0.000,B 0.000,C 90.000,E1 88.912} C_DIS
LIN {X 0.317,Y -661.078,Z 503.291,A 0.000,B 0.000,C 90.000,E1 88.396} C_DIS
LIN {X -0.019,Y -660.439,Z 503.289,A 0.000,B 0.000,C 90.000,E1 87.936} C_DIS
LIN {X 0.096,Y -659.066,Z 503.284,A 0.000,B 0.000,C 90.000,E1 87.192} C_DIS
LIN {X -0.242,Y -657.993,Z 503.282,A 0.000,B 0.000,C 90.000,E1 86.731} C_DIS
LIN {X 0.034,Y -656.665,Z 503.279,A 0.000,B 0.000,C 90.000,E1 86.216} C_DIS
LIN {X 0.142,Y -654.243,Z 503.275,A 0.000,B 0.000,C 90.000,E1 85.469} C_DIS
LIN {X -0.214,Y -652.434,Z 503.272,A 0.000,B 0.000,C 90.000,E1 85.008} C_DIS
LIN {X 0.071,Y -650.459,Z 503.269,A 0.000,B 0.000,C 90.000,E1 84.489} C_DIS
LIN {X 0.118,Y -647.118,Z 503.265,A 0.000,B 0.000,C 90.000,E1 83.742} C_DIS
LIN {X 0.241,Y -643.979,Z 503.262,A 0.000,B 0.000,C 90.000,E1 83.109} C_DIS
LIN {X -0.220,Y -640.539,Z 503.258,A 0.000,B 0.000,C 90.000,E1 82.527} C_DIS
LIN {X -0.155,Y -636.836,Z 503.255,A 0.000,B 0.000,C 90.000,E1 81.894} C_DIS
LIN {X -0.032,Y -632.738,Z 503.251,A 0.000,B 0.000,C 90.000,E1 81.254} C_DIS
LIN {X 0.232,Y -628.567,Z 503.248,A 0.000,B 0.000,C 90.000,E1 80.622} C_DIS
LIN {X 0.283,Y -623.878,Z 503.245,A 0.000,B 0.000,C 90.000,E1 79.982} C_DIS
LIN {X -0.316,Y -618.956,Z 503.241,A 0.000,B 0.000,C 90.000,E1 79.398} C_DIS
LIN {X 0.260,Y -613.559,Z 503.237,A 0.000,B 0.000,C 90.000,E1 78.701} C_DIS
LIN {X -0.227,Y -608.968,Z 503.235,A 0.000,B 0.000,C 90.000,E1 78.229} C_DIS
LIN {X -0.217,Y -602.799,Z 503.231,A 0.000,B 0.000,C 90.000,E1 77.589} C_DIS
LIN {X 0.123,Y -597.585,Z 503.228,A 0.000,B 0.000,C 90.000,E1 77.061} C_DIS
LIN {X 0.110,Y -592.018,Z 503.226,A 0.000,B 0.000,C 90.000,E1 76.589} C_DIS
LIN {X 0.328,Y -584.744,Z 503.222,A 0.000,B 0.000,C 90.000,E1 75.992} C_DIS
LIN {X -0.066,Y -581.815,Z 503.221,A 0.000,B 0.000,C 90.000,E1 75.811} C_DIS
LIN {X -0.193,Y -575.471,Z 503.219,A 0.000,B 0.000,C 90.000,E1 75.408} C_DIS
LIN {X -0.209,Y -568.991,Z 503.217,A 0.000,B 0.000,C 90.000,E1 75.046} C_DIS
LIN {X 0.018,Y -563.622,Z 503.215,A 0.000,B 0.000,C 90.000,E1 74.755} C_DIS
LIN {X 0.020,Y -558.374,Z 503.214,A 0.000,B 0.000,C 90.000,E1 74.519} C_DIS
LIN {X 0.271,Y -550.889,Z 503.212,A 0.000,B 0.000,C 90.000,E1 74.212} C_DIS
LIN {X 0.124,Y -545.133,Z 503.211,A 0.000,B 0.000,C 90.000,E1 74.047} C_DIS
LIN {X 0.032,Y -537.592,Z 503.210,A 0.000,B 0.000,C 90.000,E1 73.866} C_DIS
LIN {X 0.008,Y -531.758,Z 503.210,A 0.000,B 0.000,C 90.000,E1 73.740} C_DIS
LIN {X 0.087,Y -525.082,Z 503.209,A 0.000,B 0.000,C 90.000,E1 73.630} C_DIS
LIN {X 0.141,Y -510.725,Z 503.208,A 0.000,B 0.000,C 90.000,E1 73.449} C_DIS
LIN {X -0.174,Y -498.840,Z 503.208,A 0.000,B 0.000,C 90.000,E1 73.378} C_DIS
LIN {X 0.037,Y -494.406,Z 503.207,A 0.000,B 0.000,C 90.000,E1 73.323} C_DIS
LIN {X -0.127,Y -486.830,Z 503.207,A 0.000,B 0.000,C 90.000,E1 73.323} C_DIS
LIN {X -0.155,Y -476.306,Z 503.207,A 0.000,B 0.000,C 90.000,E1 73.268} C_DIS
LIN {X -0.190,Y -475.392,Z 503.207,A 0.000,B 0.000,C 90.000,E1 73.268} C_DIS
LIN {X -0.034,Y -474.253,Z 503.201,A 0.000,B 0.000,C 90.000,E1 72.181} C_DIS
LIN {X -0.067,Y -473.779,Z 503.199,A 0.000,B 0.000,C 90.000,E1 71.873} C_DIS
LIN {X -0.104,Y -466.209,Z 503.175,A 0.000,B 0.000,C 90.000,E1 67.486} C_DIS
LIN {X -0.162,Y -465.782,Z 503.173,A 0.000,B 0.000,C 90.000,E1 67.177} C_DIS
LIN {X -0.100,Y -464.418,Z 503.170,A 0.000,B 0.000,C 90.000,E1 66.538} C_DIS
LIN {X -0.163,Y -456.269,Z 503.147,A 0.000,B 0.000,C 90.000,E1 62.410} C_DIS
LIN {X -0.165,Y -455.120,Z 503.143,A 0.000,B 0.000,C 90.000,E1 61.769} C_DIS
LIN {X 0.150,Y -449.201,Z 503.129,A 0.000,B 0.000,C 90.000,E1 59.203} C_DIS
LIN {X 0.111,Y -449.211,Z 503.129,A 0.000,B 0.000,C 90.000,E1 59.203} C_DIS
LIN {X 0.185,Y -451.565,Z 503.126,A 0.000,B 0.000,C 90.000,E1 58.663} C_DIS
LIN {X -0.021,Y -454.290,Z 503.122,A 0.000,B 0.000,C 90.000,E1 58.043} C_DIS
LIN {X -0.083,Y -457.524,Z 503.118,A 0.000,B 0.000,C 90.000,E1 57.248} C_DIS
LIN {X 0.140,Y -459.949,Z 503.114,A 0.000,B 0.000,C 90.000,E1 56.580} C_DIS
LIN {X -0.008,Y -462.134,Z 503.111,A 0.000,B 0.000,C 90.000,E1 55.960} C_DIS
LIN {X -0.127,Y -464.958,Z 503.106,A 0.000,B 0.000,C 90.000,E1 55.022} C_DIS
LIN {X 0.143,Y -466.639,Z 503.102,A 0.000,B 0.000,C 90.000,E1 54.356} C_DIS
LIN {X 0.082,Y -468.759,Z 503.097,A 0.000,B 0.000,C 90.000,E1 53.417} C_DIS
LIN {X 0.277,Y -470.006,Z 503.093,A 0.000,B 0.000,C 90.000,E1 52.763} C_DIS
LIN {X 0.038,Y -472.016,Z 503.086,A 0.000,B 0.000,C 90.000,E1 51.537} C_DIS
LIN {X 0.121,Y -473.634,Z 503.079,A 0.000,B 0.000,C 90.000,E1 50.275} C_DIS
LIN {X 0.228,Y -474.863,Z 503.073,A 0.000,B 0.000,C 90.000,E1 49.013} C_DIS
LIN {X 0.206,Y -475.637,Z 503.067,A 0.000,B 0.000,C 90.000,E1 48.081} C_DIS
LIN {X 0.195,Y -476.250,Z 503.062,A 0.000,B 0.000,C 90.000,E1 47.148} C_DIS
LIN {X 0.190,Y -476.735,Z 503.057,A 0.000,B 0.000,C 90.000,E1 46.215} C_DIS
LIN {X -0.153,Y -477.102,Z 503.052,A 0.000,B 0.000,C 90.000,E1 45.324} C_DIS
LIN {X 0.295,Y -477.408,Z 503.045,A 0.000,B 0.000,C 90.000,E1 44.028} C_DIS
LIN {X -0.260,Y -477.429,Z 503.038,A 0.000,B 0.000,C 90.000,E1 42.852} C_DIS
LIN {X -0.142,Y -477.136,Z 503.031,A 0.000,B 0.000,C 90.000,E1 41.595} C_DIS
LIN {X 0.220,Y -476.807,Z 503.026,A 0.000,B 0.000,C 90.000,E1 40.620} C_DIS
LIN {X -0.202,Y -476.146,Z 503.017,A 0.000,B 0.000,C 90.000,E1 39.116} C_DIS
LIN {X -0.102,Y -475.175,Z 503.007,A 0.000,B 0.000,C 90.000,E1 37.237} C_DIS
LIN {X -0.033,Y -474.017,Z 502.996,A 0.000,B 0.000,C 90.000,E1 35.358} C_DIS
LIN {X -0.114,Y -473.142,Z 502.990,A 0.000,B 0.000,C 90.000,E1 34.119} C_DIS
LIN {X 0.142,Y -471.670,Z 502.979,A 0.000,B 0.000,C 90.000,E1 32.212} C_DIS
LIN {X -0.222,Y -470.615,Z 502.972,A 0.000,B 0.000,C 90.000,E1 31.003} C_DIS
LIN {X -0.032,Y -469.203,Z 502.963,A 0.000,B 0.000,C 90.000,E1 29.411} C_DIS
LIN {X -0.099,Y -467.817,Z 502.955,A 0.000,B 0.000,C 90.000,E1 27.847} C_DIS
LIN {X -0.125,Y -465.976,Z 502.942,A 0.000,B 0.000,C 90.000,E1 25.643} C_DIS
LIN {X 0.030,Y -463.713,Z 502.925,A 0.000,B 0.000,C 90.000,E1 22.461} C_DIS
LIN {X 0.052,Y -462.620,Z 502.914,A 0.000,B 0.000,C 90.000,E1 20.556} C_DIS
LIN {X -0.110,Y -461.691,Z 502.904,A 0.000,B 0.000,C 90.000,E1 18.671} C_DIS
LIN {X -0.176,Y -460.668,Z 502.890,A 0.000,B 0.000,C 90.000,E1 16.134} C_DIS
LIN {X 0.099,Y -460.125,Z 502.879,A 0.000,B 0.000,C 90.000,E1 14.189} C_DIS
LIN {X -0.054,Y -459.765,Z 502.865,A 0.000,B 0.000,C 90.000,E1 11.658} C_DIS
LIN {X 0.103,Y -459.779,Z 502.854,A 0.000,B 0.000,C 90.000,E1 9.726} C_DIS
LIN {X -0.142,Y -460.017,Z 502.845,A 0.000,B 0.000,C 90.000,E1 8.163} C_DIS
LIN {X 0.019,Y -460.414,Z 502.836,A 0.000,B 0.000,C 90.000,E1 6.549} C_DIS
LIN {X -0.061,Y -461.520,Z 502.822,A 0.000,B 0.000,C 90.000,E1 4.012} C_DIS
LIN {X -0.006,Y -463.328,Z 502.806,A 0.000,B 0.000,C 90.000,E1 1.146} C_DIS
LIN {X -0.118,Y -466.571,Z 502.787,A 0.000,B 0.000,C 90.000,E1 357.593} C_DIS
LIN {X 0.108,Y -468.288,Z 502.778,A 0.000,B 0.000,C 90.000,E1 355.988} C_DIS
LIN {X 0.008,Y -471.032,Z 502.766,A 0.000,B 0.000,C 90.000,E1 353.799} C_DIS
LIN {X 0.219,Y -473.438,Z 502.755,A 0.000,B 0.000,C 90.000,E1 351.894} C_DIS
LIN {X -0.084,Y -477.872,Z 502.738,A 0.000,B 0.000,C 90.000,E1 348.814} C_DIS
LIN {X 0.212,Y -482.679,Z 502.722,A 0.000,B 0.000,C 90.000,E1 345.992} C_DIS
LIN {X -0.019,Y -487.506,Z 502.709,A 0.000,B 0.000,C 90.000,E1 343.559} C_DIS
LIN {X 0.172,Y -492.661,Z 502.695,A 0.000,B 0.000,C 90.000,E1 341.094} C_DIS
LIN {X 0.269,Y -496.614,Z 502.685,A 0.000,B 0.000,C 90.000,E1 339.263} C_DIS
LIN {X -0.144,Y -499.245,Z 502.678,A 0.000,B 0.000,C 90.000,E1 338.103} C_DIS
LIN {X -0.265,Y -502.398,Z 502.670,A 0.000,B 0.000,C 90.000,E1 336.613} C_DIS
LIN {X 0.250,Y -504.876,Z 502.663,A 0.000,B 0.000,C 90.000,E1 335.357} C_DIS
LIN {X -0.068,Y -509.046,Z 502.652,A 0.000,B 0.000,C 90.000,E1 333.307} C_DIS
LIN {X -0.028,Y -512.095,Z 502.643,A 0.000,B 0.000,C 90.000,E1 331.820} C_DIS
LIN {X -0.028,Y -515.744,Z 502.634,A 0.000,B 0.000,C 90.000,E1 330.049} C_DIS
LIN {X 0.037,Y -519.563,Z 502.624,A 0.000,B 0.000,C 90.000,E1 328.280} C_DIS
LIN {X 0.236,Y -524.013,Z 502.612,A 0.000,B 0.000,C 90.000,E1 326.215} C_DIS
LIN {X 0.125,Y -528.579,Z 502.601,A 0.000,B 0.000,C 90.000,E1 324.196} C_DIS
LIN {X 0.029,Y -531.835,Z 502.593,A 0.000,B 0.000,C 90.000,E1 322.763} C_DIS
LIN {X -0.013,Y -535.051,Z 502.585,A 0.000,B 0.000,C 90.000,E1 321.331} C_DIS
LIN {X -0.077,Y -538.851,Z 502.576,A 0.000,B 0.000,C 90.000,E1 319.622} C_DIS
LIN {X -0.113,Y -542.661,Z 502.566,A 0.000,B 0.000,C 90.000,E1 317.919} C_DIS
LIN {X -0.062,Y -546.431,Z 502.557,A 0.000,B 0.000,C 90.000,E1 316.215} C_DIS
LIN {X 0.026,Y -549.446,Z 502.549,A 0.000,B 0.000,C 90.000,E1 314.798} C_DIS
LIN {X -0.253,Y -551.774,Z 502.543,A 0.000,B 0.000,C 90.000,E1 313.704} C_DIS
LIN {X -0.064,Y -554.736,Z 502.535,A 0.000,B 0.000,C 90.000,E1 312.285} C_DIS
LIN {X -0.044,Y -558.876,Z 502.524,A 0.000,B 0.000,C 90.000,E1 310.334} C_DIS
LIN {X -0.015,Y -562.371,Z 502.515,A 0.000,B 0.000,C 90.000,E1 308.669} C_DIS
LIN {X -0.064,Y -566.484,Z 502.504,A 0.000,B 0.000,C 90.000,E1 306.744} C_DIS
LIN {X -0.131,Y -570.002,Z 502.495,A 0.000,B 0.000,C 90.000,E1 305.105} C_DIS
LIN {X 0.015,Y -573.537,Z 502.486,A 0.000,B 0.000,C 90.000,E1 303.452} C_DIS
LIN {X 0.093,Y -576.467,Z 502.478,A 0.000,B 0.000,C 90.000,E1 302.084} C_DIS
LIN {X 0.065,Y -578.733,Z 502.472,A 0.000,B 0.000,C 90.000,E1 301.003} C_DIS
LIN {X -0.080,Y -581.394,Z 502.465,A 0.000,B 0.000,C 90.000,E1 299.667} C_DIS
LIN {X 0.190,Y -584.424,Z 502.456,A 0.000,B 0.000,C 90.000,E1 298.025} C_DIS
LIN {X -0.307,Y -586.079,Z 502.450,A 0.000,B 0.000,C 90.000,E1 297.001} C_DIS
LIN {X 0.007,Y -587.498,Z 502.444,A 0.000,B 0.000,C 90.000,E1 295.899} C_DIS
LIN {X 0.077,Y -588.692,Z 502.438,A 0.000,B 0.000,C 90.000,E1 294.823} C_DIS
LIN {X -0.075,Y -589.549,Z 502.432,A 0.000,B 0.000,C 90.000,E1 293.770} C_DIS
LIN {X 0.116,Y -590.537,Z 502.423,A 0.000,B 0.000,C 90.000,E1 292.153} C_DIS
LIN {X -0.120,Y -591.346,Z 502.416,A 0.000,B 0.000,C 90.000,E1 290.844} C_DIS
LIN {X -0.009,Y -592.015,Z 502.408,A 0.000,B 0.000,C 90.000,E1 289.504} C_DIS
LIN {X 0.235,Y -592.351,Z 502.402,A 0.000,B 0.000,C 90.000,E1 288.417} C_DIS
LIN {X 0.174,Y -592.642,Z 502.395,A 0.000,B 0.000,C 90.000,E1 287.094} C_DIS
LIN {X -0.048,Y -592.846,Z 502.388,A 0.000,B 0.000,C 90.000,E1 285.788} C_DIS
LIN {X 0.041,Y -593.007,Z 502.382,A 0.000,B 0.000,C 90.000,E1 284.717} C_DIS
LIN {X -0.208,Y -593.076,Z 502.372,A 0.000,B 0.000,C 90.000,E1 282.883} C_DIS
LIN {X 0.286,Y -593.046,Z 502.363,A 0.000,B 0.000,C 90.000,E1 281.243} C_DIS
LIN {X 0.080,Y -592.887,Z 502.354,A 0.000,B 0.000,C 90.000,E1 279.670} C_DIS
LIN {X 0.091,Y -592.628,Z 502.346,A 0.000,B 0.000,C 90.000,E1 278.341} C_DIS
LIN {X 0.178,Y -592.219,Z 502.339,A 0.000,B 0.000,C 90.000,E1 277.004} C_DIS
LIN {X -0.088,Y -591.801,Z 502.333,A 0.000,B 0.000,C 90.000,E1 275.967} C_DIS
LIN {X 0.038,Y -590.872,Z 502.324,A 0.000,B 0.000,C 90.000,E1 274.359} C_DIS
LIN {X -0.055,Y -589.873,Z 502.317,A 0.000,B 0.000,C 90.000,E1 273.037} C_DIS
LIN {X 0.164,Y -588.832,Z 502.311,A 0.000,B 0.000,C 90.000,E1 271.949} C_DIS
LIN {X -0.195,Y -587.718,Z 502.305,A 0.000,B 0.000,C 90.000,E1 270.917} C_DIS
LIN {X -0.199,Y -585.743,Z 502.296,A 0.000,B 0.000,C 90.000,E1 269.312} C_DIS
LIN {X 0.170,Y -584.005,Z 502.289,A 0.000,B 0.000,C 90.000,E1 267.936} C_DIS
LIN {X -0.071,Y -582.174,Z 502.281,A 0.000,B 0.000,C 90.000,E1 266.617} C_DIS
LIN {X 0.064,Y -580.727,Z 502.275,A 0.000,B 0.000,C 90.000,E1 265.527} C_DIS
LIN {X 0.223,Y -579.136,Z 502.269,A 0.000,B 0.000,C 90.000,E1 264.432} C_DIS
LIN {X 0.135,Y -576.450,Z 502.260,A 0.000,B 0.000,C 90.000,E1 262.818} C_DIS
LIN {X 0.173,Y -573.226,Z 502.250,A 0.000,B 0.000,C 90.000,E1 260.914} C_DIS
LIN {X 0.112,Y -570.495,Z 502.241,A 0.000,B 0.000,C 90.000,E1 259.285} C_DIS
LIN {X -0.271,Y -566.928,Z 502.230,A 0.000,B 0.000,C 90.000,E1 257.409} C_DIS
LIN {X 0.165,Y -564.286,Z 502.222,A 0.000,B 0.000,C 90.000,E1 255.992} C_DIS
LIN {X 0.010,Y -561.463,Z 502.215,A 0.000,B 0.000,C 90.000,E1 254.629} C_DIS
LIN {X -0.204,Y -558.461,Z 502.207,A 0.000,B 0.000,C 90.000,E1 253.268} C_DIS
LIN {X -0.145,Y -555.169,Z 502.199,A 0.000,B 0.000,C 90.000,E1 251.873} C_DIS
LIN {X -0.171,Y -553.188,Z 502.195,A 0.000,B 0.000,C 90.000,E1 251.040} C_DIS
LIN {X -0.016,Y -549.559,Z 502.187,A 0.000,B 0.000,C 90.000,E1 249.625} C_DIS
LIN {X 0.133,Y -545.042,Z 502.177,A 0.000,B 0.000,C 90.000,E1 247.922} C_DIS
LIN {X -0.150,Y -541.054,Z 502.170,A 0.000,B 0.000,C 90.000,E1 246.538} C_DIS
LIN {X 0.268,Y -537.699,Z 502.163,A 0.000,B 0.000,C 90.000,E1 245.357} C_DIS
LIN {X 0.285,Y -532.516,Z 502.154,A 0.000,B 0.000,C 90.000,E1 243.640} C_DIS
LIN {X -0.037,Y -527.143,Z 502.144,A 0.000,B 0.000,C 90.000,E1 241.948} C_DIS
LIN {X -0.014,Y -521.686,Z 502.135,A 0.000,B 0.000,C 90.000,E1 240.205} C_DIS
LIN {X 0.024,Y -517.208,Z 502.126,A 0.000,B 0.000,C 90.000,E1 238.742} C_DIS
LIN {X -0.106,Y -513.506,Z 502.120,A 0.000,B 0.000,C 90.000,E1 237.582} C_DIS
LIN {X 0.050,Y -508.714,Z 502.112,A 0.000,B 0.000,C 90.000,E1 236.087} C_DIS
LIN {X -0.020,Y -503.907,Z 502.103,A 0.000,B 0.000,C 90.000,E1 234.609} C_DIS
LIN {X 0.274,Y -497.251,Z 502.092,A 0.000,B 0.000,C 90.000,E1 232.477} C_DIS
LIN {X -0.017,Y -489.259,Z 502.077,A 0.000,B 0.000,C 90.000,E1 229.784} C_DIS
LIN {X 0.050,Y -483.400,Z 502.065,A 0.000,B 0.000,C 90.000,E1 227.634} C_DIS
LIN {X -0.055,Y -477.624,Z 502.053,A 0.000,B 0.000,C 90.000,E1 225.486} C_DIS
LIN {X 0.021,Y -472.117,Z 502.041,A 0.000,B 0.000,C 90.000,E1 223.299} C_DIS
LIN {X -0.113,Y -467.549,Z 502.030,A 0.000,B 0.000,C 90.000,E1 221.434} C_DIS
LIN {X -0.148,Y -461.844,Z 502.016,A 0.000,B 0.000,C 90.000,E1 218.910} C_DIS
LIN {X -0.009,Y -457.029,Z 502.004,A 0.000,B 0.000,C 90.000,E1 216.664} C_DIS
LIN {X 0.001,Y -453.129,Z 501.993,A 0.000,B 0.000,C 90.000,E1 214.739} C_DIS
LIN {X 0.181,Y -448.129,Z 501.979,A 0.000,B 0.000,C 90.000,E1 212.133} C_DIS
LIN {X -0.006,Y -444.531,Z 501.968,A 0.000,B 0.000,C 90.000,E1 210.207} C_DIS
LIN {X 0.112,Y -440.949,Z 501.957,A 0.000,B 0.000,C 90.000,E1 208.231} C_DIS
LIN {X 0.067,Y -438.629,Z 501.950,A 0.000,B 0.000,C 90.000,E1 206.924} C_DIS
LIN {X 0.175,Y -436.300,Z 501.942,A 0.000,B 0.000,C 90.000,E1 205.591} C_DIS
LIN {X -0.105,Y -432.853,Z 501.931,A 0.000,B 0.000,C 90.000,E1 203.643} C_DIS
LIN {X -0.075,Y -429.508,Z 501.920,A 0.000,B 0.000,C 90.000,E1 201.642} C_DIS
LIN {X 0.157,Y -426.873,Z 501.911,A 0.000,B 0.000,C 90.000,E1 199.939} C_DIS
LIN {X -0.032,Y -422.979,Z 501.896,A 0.000,B 0.000,C 90.000,E1 197.275} C_DIS
LIN {X 0.047,Y -419.874,Z 501.883,A 0.000,B 0.000,C 90.000,E1 194.898} C_DIS
LIN {X -0.060,Y -417.015,Z 501.870,A 0.000,B 0.000,C 90.000,E1 192.535} C_DIS
LIN {X -0.020,Y -414.356,Z 501.856,A 0.000,B 0.000,C 90.000,E1 190.141} C_DIS
LIN {X -0.167,Y -412.166,Z 501.845,A 0.000,B 0.000,C 90.000,E1 188.106} C_DIS
LIN {X -0.072,Y -410.138,Z 501.833,A 0.000,B 0.000,C 90.000,E1 186.030} C_DIS
LIN {X -0.033,Y -408.067,Z 501.822,A 0.000,B 0.000,C 90.000,E1 183.955} C_DIS
LIN {X -0.157,Y -405.862,Z 501.807,A 0.000,B 0.000,C 90.000,E1 181.203} C_DIS
LIN {X 0.071,Y -404.372,Z 501.793,A 0.000,B 0.000,C 90.000,E1 178.740} C_DIS
LIN {X 0.129,Y -402.756,Z 501.770,A 0.000,B 0.000,C 90.000,E1 174.552} C_DIS
LIN {X -0.020,Y -402.465,Z 501.752,A 0.000,B 0.000,C 90.000,E1 171.432} C_DIS
LIN {X -0.045,Y -402.698,Z 501.739,A 0.000,B 0.000,C 90.000,E1 168.993} C_DIS
LIN {X 0.085,Y -403.281,Z 501.725,A 0.000,B 0.000,C 90.000,E1 166.533} C_DIS
LIN {X 0.232,Y -404.470,Z 501.708,A 0.000,B 0.000,C 90.000,E1 163.378} C_DIS
LIN {X 0.179,Y -406.006,Z 501.692,A 0.000,B 0.000,C 90.000,E1 160.604} C_DIS
LIN {X -0.148,Y -406.935,Z 501.685,A 0.000,B 0.000,C 90.000,E1 159.263} C_DIS
LIN {X 0.179,Y -408.805,Z 501.671,A 0.000,B 0.000,C 90.000,E1 156.794} C_DIS
LIN {X -0.035,Y -410.902,Z 501.658,A 0.000,B 0.000,C 90.000,E1 154.409} C_DIS
LIN {X 0.127,Y -412.484,Z 501.648,A 0.000,B 0.000,C 90.000,E1 152.666} C_DIS
LIN {X -0.040,Y -413.957,Z 501.639,A 0.000,B 0.000,C 90.000,E1 150.973} C_DIS
LIN {X -0.030,Y -415.631,Z 501.627,A 0.000,B 0.000,C 90.000,E1 148.918} C_DIS
LIN {X 0.109,Y -416.740,Z 501.620,A 0.000,B 0.000,C 90.000,E1 147.533} C_DIS
LIN {X -0.268,Y -418.017,Z 501.610,A 0.000,B 0.000,C 90.000,E1 145.881} C_DIS
LIN {X 0.202,Y -419.261,Z 501.601,A 0.000,B 0.000,C 90.000,E1 144.116} C_DIS
LIN {X -0.020,Y -420.666,Z 501.590,A 0.000,B 0.000,C 90.000,E1 142.110} C_DIS
LIN {X -0.167,Y -421.800,Z 501.580,A 0.000,B 0.000,C 90.000,E1 140.436} C_DIS
LIN {X 0.032,Y -422.592,Z 501.573,A 0.000,B 0.000,C 90.000,E1 139.057} C_DIS
LIN {X -0.033,Y -423.315,Z 501.565,A 0.000,B 0.000,C 90.000,E1 137.715} C_DIS
LIN {X -0.023,Y -423.674,Z 501.559,A 0.000,B 0.000,C 90.000,E1 136.701} C_DIS
LIN {X -0.012,Y -423.968,Z 501.554,A 0.000,B 0.000,C 90.000,E1 135.688} C_DIS
LIN {X -0.002,Y -424.218,Z 501.548,A 0.000,B 0.000,C 90.000,E1 134.676} C_DIS
LIN {X 0.021,Y -424.313,Z 501.543,A 0.000,B 0.000,C 90.000,E1 133.662} C_DIS
LIN {X -0.263,Y -424.158,Z 501.537,A 0.000,B 0.000,C 90.000,E1 132.690} C_DIS
LIN {X -0.025,Y -423.547,Z 501.530,A 0.000,B 0.000,C 90.000,E1 131.310} C_DIS
LIN {X 0.199,Y -422.654,Z 501.522,A 0.000,B 0.000,C 90.000,E1 129.930} C_DIS
LIN {X 0.078,Y -421.084,Z 501.513,A 0.000,B 0.000,C 90.000,E1 128.257} C_DIS
LIN {X -0.019,Y -419.754,Z 501.505,A 0.000,B 0.000,C 90.000,E1 126.916} C_DIS
LIN {X 0.275,Y -418.329,Z 501.498,A 0.000,B 0.000,C 90.000,E1 125.518} C_DIS
LIN {X 0.034,Y -417.728,Z 501.495,A 0.000,B 0.000,C 90.000,E1 125.025} C_DIS
LIN {X -0.005,Y -417.738,Z 501.495,A 0.000,B 0.000,C 90.000,E1 125.025} C_DIS
LIN {X 0.188,Y -427.104,Z 501.475,A 0.000,B 0.000,C 90.000,E1 121.465} C_DIS
LIN {X 0.160,Y -430.156,Z 501.469,A 0.000,B 0.000,C 90.000,E1 120.463} C_DIS
LIN {X 0.159,Y -431.086,Z 501.468,A 0.000,B 0.000,C 90.000,E1 120.129} C_DIS
LIN {X 0.106,Y -440.180,Z 501.447,A 0.000,B 0.000,C 90.000,E1 116.488} C_DIS
LIN {X 0.113,Y -444.942,Z 501.438,A 0.000,B 0.000,C 90.000,E1 114.847} C_DIS
LIN {X -0.034,Y -454.063,Z 501.417,A 0.000,B 0.000,C 90.000,E1 110.972} C_DIS
LIN {X 0.079,Y -456.716,Z 501.411,A 0.000,B 0.000,C 90.000,E1 109.993} C_DIS
LIN {X -0.021,Y -457.501,Z 501.409,A 0.000,B 0.000,C 90.000,E1 109.685} C_DIS
LIN {X 0.239,Y -461.756,Z 501.397,A 0.000,B 0.000,C 90.000,E1 107.457} C_DIS
LIN {X 0.199,Y -461.799,Z 501.397,A 0.000,B 0.000,C 90.000,E1 107.457} C_DIS
LIN {X 0.176,Y -477.697,Z 501.395,A 0.000,B 0.000,C 90.000,E1 107.094} C_DIS
LIN {X -0.062,Y -488.346,Z 501.394,A 0.000,B 0.000,C 90.000,E1 106.858} C_DIS
LIN {X 0.023,Y -498.828,Z 501.392,A 0.000,B 0.000,C 90.000,E1 106.567} C_DIS
LIN {X 0.096,Y -509.648,Z 501.390,A 0.000,B 0.000,C 90.000,E1 106.260} C_DIS
LIN {X -0.096,Y -520.005,Z 501.389,A 0.000,B 0.000,C 90.000,E1 105.969} C_DIS
LIN {X 0.131,Y -530.411,Z 501.387,A 0.000,B 0.000,C 90.000,E1 105.607} C_DIS
LIN {X 0.198,Y -540.502,Z 501.385,A 0.000,B 0.000,C 90.000,E1 105.245} C_DIS
LIN {X -0.037,Y -547.133,Z 501.383,A 0.000,B 0.000,C 90.000,E1 105.009} C_DIS
LIN {X 0.057,Y -553.619,Z 501.382,A 0.000,B 0.000,C 90.000,E1 104.717} C_DIS
LIN {X 0.068,Y -560.163,Z 501.380,A 0.000,B 0.000,C 90.000,E1 104.411} C_DIS
LIN {X 0.248,Y -566.195,Z 501.378,A 0.000,B 0.000,C 90.000,E1 104.064} C_DIS
LIN {X 0.159,Y -572.087,Z 501.376,A 0.000,B 0.000,C 90.000,E1 103.716} C_DIS
LIN {X -0.213,Y -576.624,Z 501.375,A 0.000,B 0.000,C 90.000,E1 103.467} C_DIS
LIN {X -0.108,Y -578.358,Z 501.374,A 0.000,B 0.000,C 90.000,E1 103.355} C_DIS
LIN {X 0.052,Y -585.290,Z 501.371,A 0.000,B 0.000,C 90.000,E1 102.827} C_DIS
LIN {X 0.153,Y -590.393,Z 501.369,A 0.000,B 0.000,C 90.000,E1 102.411} C_DIS
LIN {X 0.055,Y -596.012,Z 501.366,A 0.000,B 0.000,C 90.000,E1 101.951} C_DIS
LIN {X -0.162,Y -602.512,Z 501.363,A 0.000,B 0.000,C 90.000,E1 101.366} C_DIS
LIN {X 0.093,Y -608.701,Z 501.360,A 0.000,B 0.000,C 90.000,E1 100.715} C_DIS
LIN {X 0.133,Y -613.490,Z 501.357,A 0.000,B 0.000,C 90.000,E1 100.197} C_DIS
LIN {X 0.085,Y -619.036,Z 501.353,A 0.000,B 0.000,C 90.000,E1 99.557} C_DIS
LIN {X 0.171,Y -625.047,Z 501.349,A 0.000,B 0.000,C 90.000,E1 98.803} C_DIS
LIN {X -0.101,Y -631.338,Z 501.344,A 0.000,B 0.000,C 90.000,E1 97.936} C_DIS
LIN {X 0.118,Y -634.610,Z 501.341,A 0.000,B 0.000,C 90.000,E1 97.409} C_DIS
LIN {X 0.007,Y -639.168,Z 501.337,A 0.000,B 0.000,C 90.000,E1 96.663} C_DIS
LIN {X 0.016,Y -643.169,Z 501.333,A 0.000,B 0.000,C 90.000,E1 95.910} C_DIS
LIN {X 0.348,Y -648.645,Z 501.327,A 0.000,B 0.000,C 90.000,E1 94.759} C_DIS
LIN {X -0.274,Y -651.970,Z 501.323,A 0.000,B 0.000,C 90.000,E1 94.069} C_DIS
LIN {X -0.049,Y -654.002,Z 501.320,A 0.000,B 0.000,C 90.000,E1 93.555} C_DIS
LIN {X 0.031,Y -656.583,Z 501.316,A 0.000,B 0.000,C 90.000,E1 92.808} C_DIS
LIN {X 0.297,Y -658.090,Z 501.313,A 0.000,B 0.000,C 90.000,E1 92.293} C_DIS
LIN {X -0.079,Y -659.302,Z 501.310,A 0.000,B 0.000,C 90.000,E1 91.835} C_DIS
LIN {X 0.046,Y -660.620,Z 501.306,A 0.000,B 0.000,C 90.000,E1 91.088} C_DIS
LIN {X -0.314,Y -661.214,Z 501.303,A 0.000,B 0.000,C 90.000,E1 90.630} C_DIS
LIN {X -0.007,Y -661.623,Z 501.301,A 0.000,B 0.000,C 90.000,E1 90.115} C_DIS
LIN {X 0.301,Y -661.652,Z 501.298,A 0.000,B 0.000,C 90.000,E1 89.599} C_DIS
LIN {X -0.227,Y -661.331,Z 501.294,A 0.000,B 0.000,C 90.000,E1 88.912} C_DIS
LIN {X 0.077,Y -660.872,Z 501.291,A 0.000,B 0.000,C 90.000,E1 88.396} C_DIS
LIN {X -0.260,Y -660.196,Z 501.288,A 0.000,B 0.000,C 90.000,E1 87.936} C_DIS
LIN {X -0.146,Y -658.762,Z 501.284,A 0.000,B 0.000,C 90.000,E1 87.192} C_DIS
LIN {X -0.019,Y -656.935,Z 501.280,A 0.000,B 0.000,C 90.000,E1 86.445} C_DIS
LIN {X 0.246,Y -655.374,Z 501.278,A 0.000,B 0.000,C 90.000,E1 85.931} C_DIS
LIN {X -0.314,Y -652.805,Z 501.273,A 0.000,B 0.000,C 90.000,E1 85.241} C_DIS
LIN {X -0.184,Y -649.742,Z 501.269,A 0.000,B 0.000,C 90.000,E1 84.489} C_DIS
LIN {X -0.030,Y -646.867,Z 501.266,A 0.000,B 0.000,C 90.000,E1 83.856} C_DIS
LIN {X 0.095,Y -643.687,Z 501.262,A 0.000,B 0.000,C 90.000,E1 83.223} C_DIS
LIN {X 0.185,Y -640.205,Z 501.259,A 0.000,B 0.000,C 90.000,E1 82.591} C_DIS
LIN {X 0.192,Y -635.629,Z 501.255,A 0.000,B 0.000,C 90.000,E1 81.837} C_DIS
LIN {X 0.302,Y -631.471,Z 501.251,A 0.000,B 0.000,C 90.000,E1 81.197} C_DIS
LIN {X -0.342,Y -626.994,Z 501.248,A 0.000,B 0.000,C 90.000,E1 80.622} C_DIS
LIN {X -0.301,Y -622.124,Z 501.244,A 0.000,B 0.000,C 90.000,E1 79.982} C_DIS
LIN {X -0.132,Y -617.956,Z 501.241,A 0.000,B 0.000,C 90.000,E1 79.454} C_DIS
LIN {X 0.012,Y -613.549,Z 501.239,A 0.000,B 0.000,C 90.000,E1 78.926} C_DIS
LIN {X 0.031,Y -607.650,Z 501.235,A 0.000,B 0.000,C 90.000,E1 78.285} C_DIS
LIN {X 0.228,Y -602.702,Z 501.232,A 0.000,B 0.000,C 90.000,E1 77.757} C_DIS
LIN {X -0.001,Y -597.453,Z 501.229,A 0.000,B 0.000,C 90.000,E1 77.285} C_DIS
LIN {X 0.084,Y -586.067,Z 501.224,A 0.000,B 0.000,C 90.000,E1 76.353} C_DIS
LIN {X -0.073,Y -579.855,Z 501.222,A 0.000,B 0.000,C 90.000,E1 75.936} C_DIS
LIN {X -0.210,Y -575.213,Z 501.220,A 0.000,B 0.000,C 90.000,E1 75.644} C_DIS
LIN {X 0.202,Y -568.383,Z 501.218,A 0.000,B 0.000,C 90.000,E1 75.227} C_DIS
LIN {X -0.207,Y -561.183,Z 501.216,A 0.000,B 0.000,C 90.000,E1 74.936} C_DIS
LIN {X -0.044,Y -555.813,Z 501.215,A 0.000,B 0.000,C 90.000,E1 74.700} C_DIS
LIN {X -0.200,Y -550.117,Z 501.214,A 0.000,B 0.000,C 90.000,E1 74.519} C_DIS
LIN {X -0.076,Y -544.378,Z 501.213,A 0.000,B 0.000,C 90.000,E1 74.338} C_DIS
LIN {X -0.161,Y -538.658,Z 501.212,A 0.000,B 0.000,C 90.000,E1 74.212} C_DIS
LIN {X 0.065,Y -530.695,Z 501.211,A 0.000,B 0.000,C 90.000,E1 74.031} C_DIS
LIN {X -0.080,Y -525.990,Z 501.211,A 0.000,B 0.000,C 90.000,E1 73.976} C_DIS
LIN {X -0.120,Y -508.438,Z 501.210,A 0.000,B 0.000,C 90.000,E1 73.795} C_DIS
LIN {X 0.091,Y -494.249,Z 501.209,A 0.000,B 0.000,C 90.000,E1 73.685} C_DIS
LIN {X -0.248,Y -480.080,Z 501.209,A 0.000,B 0.000,C 90.000,E1 73.685} C_DIS
LIN {X -0.274,Y -475.998,Z 501.209,A 0.000,B 0.000,C 90.000,E1 73.685} C_DIS
LIN {X 0.135,Y -475.865,Z 501.209,A 0.000,B 0.000,C 90.000,E1 73.630} C_DIS
LIN {X 0.074,Y -473.965,Z 501.200,A 0.000,B 0.000,C 90.000,E1 71.945} C_DIS
LIN {X 0.200,Y -466.334,Z 501.175,A 0.000,B 0.000,C 90.000,E1 67.539} C_DIS
LIN {X 0.084,Y -465.367,Z 501.172,A 0.000,B 0.000,C 90.000,E1 66.922} C_DIS
LIN {X 0.052,Y -456.958,Z 501.149,A 0.000,B 0.000,C 90.000,E1 62.794} C_DIS
LIN {X -0.052,Y -455.351,Z 501.144,A 0.000,B 0.000,C 90.000,E1 61.847} C_DIS
LIN {X -0.029,Y -449.596,Z 501.130,A 0.000,B 0.000,C 90.000,E1 59.410} C_DIS
LIN {X -0.068,Y -449.615,Z 501.130,A 0.000,B 0.000,C 90.000,E1 59.410} C_DIS
LIN {X 0.031,Y -453.155,Z 501.126,A 0.000,B 0.000,C 90.000,E1 58.614} C_DIS
LIN {X -0.079,Y -457.963,Z 501.119,A 0.000,B 0.000,C 90.000,E1 57.502} C_DIS
LIN {X 0.012,Y -462.180,Z 501.113,A 0.000,B 0.000,C 90.000,E1 56.373} C_DIS
LIN {X 0.143,Y -464.265,Z 501.110,A 0.000,B 0.000,C 90.000,E1 55.722} C_DIS
LIN {X 0.029,Y -466.137,Z 501.106,A 0.000,B 0.000,C 90.000,E1 55.102} C_DIS
LIN {X -0.072,Y -467.840,Z 501.103,A 0.000,B 0.000,C 90.000,E1 54.482} C_DIS
LIN {X -0.117,Y -469.945,Z 501.097,A 0.000,B 0.000,C 90.000,E1 53.543} C_DIS
LIN {X -0.196,Y -471.210,Z 501.094,A 0.000,B 0.000,C 90.000,E1 52.924} C_DIS
LIN {X 0.242,Y -473.171,Z 501.087,A 0.000,B 0.000,C 90.000,E1 51.618} C_DIS
LIN {X -0.111,Y -474.368,Z 501.082,A 0.000,B 0.000,C 90.000,E1 50.723} C_DIS
LIN {X 0.128,Y -475.069,Z 501.078,A 0.000,B 0.000,C 90.000,E1 50.070} C_DIS
LIN {X -0.107,Y -476.224,Z 501.071,A 0.000,B 0.000,C 90.000,E1 48.852} C_DIS
LIN {X -0.111,Y -476.917,Z 501.066,A 0.000,B 0.000,C 90.000,E1 47.919} C_DIS
LIN {X 0.005,Y -477.671,Z 501.059,A 0.000,B 0.000,C 90.000,E1 46.662} C_DIS
LIN {X 0.132,Y -478.103,Z 501.052,A 0.000,B 0.000,C 90.000,E1 45.405} C_DIS
LIN {X -0.080,Y -478.372,Z 501.046,A 0.000,B 0.000,C 90.000,E1 44.190} C_DIS
LIN {X -0.061,Y -478.423,Z 501.040,A 0.000,B 0.000,C 90.000,E1 43.257} C_DIS
LIN {X 0.077,Y -478.183,Z 501.033,A 0.000,B 0.000,C 90.000,E1 42.000} C_DIS
LIN {X -0.111,Y -477.736,Z 501.027,A 0.000,B 0.000,C 90.000,E1 40.782} C_DIS
LIN {X -0.044,Y -476.884,Z 501.016,A 0.000,B 0.000,C 90.000,E1 38.910} C_DIS
LIN {X -0.098,Y -476.061,Z 501.008,A 0.000,B 0.000,C 90.000,E1 37.363} C_DIS
LIN {X -0.080,Y -475.114,Z 500.999,A 0.000,B 0.000,C 90.000,E1 35.804} C_DIS
LIN {X 0.129,Y -474.231,Z 500.992,A 0.000,B 0.000,C 90.000,E1 34.532} C_DIS
LIN {X 0.232,Y -473.018,Z 500.983,A 0.000,B 0.000,C 90.000,E1 32.959} C_DIS
LIN {X 0.063,Y -471.757,Z 500.975,A 0.000,B 0.000,C 90.000,E1 31.416} C_DIS
LIN {X -0.130,Y -470.315,Z 500.966,A 0.000,B 0.000,C 90.000,E1 29.873} C_DIS
LIN {X 0.139,Y -468.268,Z 500.954,A 0.000,B 0.000,C 90.000,E1 27.641} C_DIS
LIN {X -0.085,Y -466.416,Z 500.941,A 0.000,B 0.000,C 90.000,E1 25.463} C_DIS
LIN {X 0.160,Y -464.347,Z 500.926,A 0.000,B 0.000,C 90.000,E1 22.589} C_DIS
LIN {X 0.129,Y -463.027,Z 500.913,A 0.000,B 0.000,C 90.000,E1 20.375} C_DIS
LIN {X -0.022,Y -462.096,Z 500.903,A 0.000,B 0.000,C 90.000,E1 18.489} C_DIS
LIN {X 0.011,Y -461.168,Z 500.890,A 0.000,B 0.000,C 90.000,E1 16.260} C_DIS
LIN {X 0.070,Y -460.693,Z 500.882,A 0.000,B 0.000,C 90.000,E1 14.662} C_DIS
LIN {X 0.033,Y -460.172,Z 500.867,A 0.000,B 0.000,C 90.000,E1 12.119} C_DIS
LIN {X -0.103,Y -460.131,Z 500.855,A 0.000,B 0.000,C 90.000,E1 9.905} C_DIS
LIN {X 0.187,Y -460.322,Z 500.846,A 0.000,B 0.000,C 90.000,E1 8.276} C_DIS
LIN {X -0.107,Y -460.670,Z 500.837,A 0.000,B 0.000,C 90.000,E1 6.720} C_DIS
LIN {X 0.014,Y -461.850,Z 500.821,A 0.000,B 0.000,C 90.000,E1 3.841} C_DIS
LIN {X -0.129,Y -463.445,Z 500.807,A 0.000,B 0.000,C 90.000,E1 1.318} C_DIS
LIN {X -0.112,Y -466.763,Z 500.787,A 0.000,B 0.000,C 90.000,E1 357.593} C_DIS
LIN {X 0.117,Y -468.479,Z 500.778,A 0.000,B 0.000,C 90.000,E1 355.988} C_DIS
LIN {X 0.023,Y -471.202,Z 500.766,A 0.000,B 0.000,C 90.000,E1 353.799} C_DIS
LIN {X 0.237,Y -473.565,Z 500.755,A 0.000,B 0.000,C 90.000,E1 351.894} C_DIS
LIN {X -0.060,Y -478.029,Z 500.738,A 0.000,B 0.000,C 90.000,E1 348.814} C_DIS
LIN {X 0.242,Y -482.896,Z 500.722,A 0.000,B 0.000,C 90.000,E1 345.992} C_DIS
LIN {X 0.018,Y -487.737,Z 500.709,A 0.000,B 0.000,C 90.000,E1 343.559} C_DIS
LIN {X 0.154,Y -491.568,Z 500.699,A 0.000,B 0.000,C 90.000,E1 341.710} C_DIS
LIN {X 0.130,Y -494.206,Z 500.692,A 0.000,B 0.000,C 90.000,E1 340.496} C_DIS
LIN {X -0.145,Y -496.910,Z 500.685,A 0.000,B 0.000,C 90.000,E1 339.316} C_DIS
LIN {X -0.024,Y -500.168,Z 500.677,A 0.000,B 0.000,C 90.000,E1 337.794} C_DIS
LIN {X -0.128,Y -503.342,Z 500.668,A 0.000,B 0.000,C 90.000,E1 336.305} C_DIS
LIN {X -0.057,Y -505.804,Z 500.662,A 0.000,B 0.000,C 90.000,E1 335.101} C_DIS
LIN {X 0.103,Y -510.045,Z 500.650,A 0.000,B 0.000,C 90.000,E1 332.999} C_DIS
LIN {X 0.156,Y -513.085,Z 500.642,A 0.000,B 0.000,C 90.000,E1 331.513} C_DIS
LIN {X -0.192,Y -516.196,Z 500.634,A 0.000,B 0.000,C 90.000,E1 330.078} C_DIS
LIN {X 0.142,Y -520.059,Z 500.624,A 0.000,B 0.000,C 90.000,E1 328.280} C_DIS
LIN {X 0.064,Y -524.551,Z 500.613,A 0.000,B 0.000,C 90.000,E1 326.246} C_DIS
LIN {X 0.258,Y -529.159,Z 500.601,A 0.000,B 0.000,C 90.000,E1 324.196} C_DIS
LIN {X 0.163,Y -533.101,Z 500.592,A 0.000,B 0.000,C 90.000,E1 322.477} C_DIS
LIN {X 0.144,Y -535.725,Z 500.585,A 0.000,B 0.000,C 90.000,E1 321.331} C_DIS
LIN {X 0.095,Y -539.551,Z 500.576,A 0.000,B 0.000,C 90.000,E1 319.622} C_DIS
LIN {X 0.077,Y -543.404,Z 500.566,A 0.000,B 0.000,C 90.000,E1 317.919} C_DIS
LIN {X -0.253,Y -546.580,Z 500.558,A 0.000,B 0.000,C 90.000,E1 316.539} C_DIS
LIN {X 0.225,Y -549.627,Z 500.551,A 0.000,B 0.000,C 90.000,E1 315.081} C_DIS
LIN {X -0.018,Y -552.592,Z 500.543,A 0.000,B 0.000,C 90.000,E1 313.704} C_DIS
LIN {X 0.249,Y -556.165,Z 500.534,A 0.000,B 0.000,C 90.000,E1 312.000} C_DIS
LIN {X -0.197,Y -559.737,Z 500.524,A 0.000,B 0.000,C 90.000,E1 310.378} C_DIS
LIN {X -0.074,Y -563.229,Z 500.515,A 0.000,B 0.000,C 90.000,E1 308.705} C_DIS
LIN {X -0.200,Y -567.383,Z 500.504,A 0.000,B 0.000,C 90.000,E1 306.790} C_DIS
LIN {X 0.208,Y -570.939,Z 500.495,A 0.000,B 0.000,C 90.000,E1 305.105} C_DIS
LIN {X -0.103,Y -574.531,Z 500.486,A 0.000,B 0.000,C 90.000,E1 303.499} C_DIS
LIN {X -0.176,Y -578.104,Z 500.477,A 0.000,B 0.000,C 90.000,E1 301.878} C_DIS
LIN {X -0.184,Y -580.351,Z 500.471,A 0.000,B 0.000,C 90.000,E1 300.797} C_DIS
LIN {X 0.202,Y -583.027,Z 500.464,A 0.000,B 0.000,C 90.000,E1 299.411} C_DIS
LIN {X -0.158,Y -585.497,Z 500.456,A 0.000,B 0.000,C 90.000,E1 298.103} C_DIS
LIN {X 0.153,Y -587.198,Z 500.450,A 0.000,B 0.000,C 90.000,E1 297.001} C_DIS
LIN {X -0.191,Y -588.285,Z 500.446,A 0.000,B 0.000,C 90.000,E1 296.232} C_DIS
LIN {X -0.213,Y -589.841,Z 500.438,A 0.000,B 0.000,C 90.000,E1 294.899} C_DIS
LIN {X 0.001,Y -590.538,Z 500.434,A 0.000,B 0.000,C 90.000,E1 294.079} C_DIS
LIN {X -0.226,Y -591.508,Z 500.426,A 0.000,B 0.000,C 90.000,E1 292.770} C_DIS
LIN {X -0.001,Y -592.542,Z 500.418,A 0.000,B 0.000,C 90.000,E1 291.153} C_DIS
LIN {X 0.132,Y -593.256,Z 500.410,A 0.000,B 0.000,C 90.000,E1 289.812} C_DIS
LIN {X 0.087,Y -593.733,Z 500.403,A 0.000,B 0.000,C 90.000,E1 288.489} C_DIS
LIN {X -0.069,Y -594.123,Z 500.394,A 0.000,B 0.000,C 90.000,E1 286.913} C_DIS
LIN {X -0.267,Y -594.372,Z 500.387,A 0.000,B 0.000,C 90.000,E1 285.607} C_DIS
LIN {X -0.160,Y -594.561,Z 500.381,A 0.000,B 0.000,C 90.000,E1 284.537} C_DIS
LIN {X -0.077,Y -594.701,Z 500.372,A 0.000,B 0.000,C 90.000,E1 282.939} C_DIS
LIN {X 0.033,Y -594.701,Z 500.362,A 0.000,B 0.000,C 90.000,E1 281.074} C_DIS
LIN {X 0.275,Y -594.597,Z 500.354,A 0.000,B 0.000,C 90.000,E1 279.726} C_DIS
LIN {X -0.277,Y -594.352,Z 500.347,A 0.000,B 0.000,C 90.000,E1 278.454} C_DIS
LIN {X -0.234,Y -593.957,Z 500.340,A 0.000,B 0.000,C 90.000,E1 277.125} C_DIS
LIN {X -0.204,Y -593.410,Z 500.332,A 0.000,B 0.000,C 90.000,E1 275.796} C_DIS
LIN {X -0.040,Y -592.421,Z 500.323,A 0.000,B 0.000,C 90.000,E1 274.188} C_DIS
LIN {X -0.104,Y -591.410,Z 500.316,A 0.000,B 0.000,C 90.000,E1 272.865} C_DIS
LIN {X -0.021,Y -589.733,Z 500.307,A 0.000,B 0.000,C 90.000,E1 271.260} C_DIS
LIN {X 0.204,Y -588.419,Z 500.301,A 0.000,B 0.000,C 90.000,E1 270.172} C_DIS
LIN {X -0.176,Y -587.071,Z 500.295,A 0.000,B 0.000,C 90.000,E1 269.141} C_DIS
LIN {X -0.181,Y -584.904,Z 500.286,A 0.000,B 0.000,C 90.000,E1 267.535} C_DIS
LIN {X -0.026,Y -582.303,Z 500.276,A 0.000,B 0.000,C 90.000,E1 265.641} C_DIS
LIN {X -0.261,Y -580.221,Z 500.268,A 0.000,B 0.000,C 90.000,E1 264.318} C_DIS
LIN {X -0.118,Y -576.956,Z 500.258,A 0.000,B 0.000,C 90.000,E1 262.413} C_DIS
LIN {X 0.022,Y -573.665,Z 500.247,A 0.000,B 0.000,C 90.000,E1 260.500} C_DIS
LIN {X 0.156,Y -571.820,Z 500.241,A 0.000,B 0.000,C 90.000,E1 259.398} C_DIS
LIN {X 0.182,Y -568.689,Z 500.232,A 0.000,B 0.000,C 90.000,E1 257.757} C_DIS
LIN {X -0.031,Y -566.004,Z 500.225,A 0.000,B 0.000,C 90.000,E1 256.408} C_DIS
LIN {X 0.228,Y -563.803,Z 500.218,A 0.000,B 0.000,C 90.000,E1 255.283} C_DIS
LIN {X 0.059,Y -560.846,Z 500.211,A 0.000,B 0.000,C 90.000,E1 253.921} C_DIS
LIN {X -0.139,Y -558.298,Z 500.205,A 0.000,B 0.000,C 90.000,E1 252.834} C_DIS
LIN {X -0.248,Y -554.959,Z 500.197,A 0.000,B 0.000,C 90.000,E1 251.456} C_DIS
LIN {X -0.098,Y -552.848,Z 500.192,A 0.000,B 0.000,C 90.000,E1 250.604} C_DIS
LIN {X -0.136,Y -549.165,Z 500.184,A 0.000,B 0.000,C 90.000,E1 249.209} C_DIS
LIN {X -0.051,Y -545.311,Z 500.177,A 0.000,B 0.000,C 90.000,E1 247.794} C_DIS
LIN {X -0.068,Y -542.090,Z 500.170,A 0.000,B 0.000,C 90.000,E1 246.666} C_DIS
LIN {X -0.126,Y -538.736,Z 500.164,A 0.000,B 0.000,C 90.000,E1 245.537} C_DIS
LIN {X -0.076,Y -533.528,Z 500.155,A 0.000,B 0.000,C 90.000,E1 243.819} C_DIS
LIN {X -0.148,Y -528.131,Z 500.145,A 0.000,B 0.000,C 90.000,E1 242.103} C_DIS
LIN {X 0.145,Y -522.657,Z 500.135,A 0.000,B 0.000,C 90.000,E1 240.333} C_DIS
LIN {X 0.201,Y -518.143,Z 500.127,A 0.000,B 0.000,C 90.000,E1 238.869} C_DIS
LIN {X 0.086,Y -514.445,Z 500.121,A 0.000,B 0.000,C 90.000,E1 237.709} C_DIS
LIN {X 0.261,Y -509.656,Z 500.113,A 0.000,B 0.000,C 90.000,E1 236.215} C_DIS
LIN {X -0.082,Y -504.816,Z 500.104,A 0.000,B 0.000,C 90.000,E1 234.769} C_DIS
LIN {X -0.168,Y -498.107,Z 500.093,A 0.000,B 0.000,C 90.000,E1 232.683} C_DIS
LIN {X 0.115,Y -489.155,Z 500.076,A 0.000,B 0.000,C 90.000,E1 229.622} C_DIS
LIN {X 0.182,Y -483.281,Z 500.064,A 0.000,B 0.000,C 90.000,E1 227.472} C_DIS
LIN {X -0.047,Y -478.314,Z 500.054,A 0.000,B 0.000,C 90.000,E1 225.648} C_DIS
LIN {X 0.048,Y -472.787,Z 500.042,A 0.000,B 0.000,C 90.000,E1 223.461} C_DIS
LIN {X -0.068,Y -468.179,Z 500.031,A 0.000,B 0.000,C 90.000,E1 221.595} C_DIS
LIN {X -0.082,Y -462.431,Z 500.017,A 0.000,B 0.000,C 90.000,E1 219.072} C_DIS
LIN {X 0.080,Y -457.619,Z 500.005,A 0.000,B 0.000,C 90.000,E1 216.824} C_DIS
LIN {X 0.109,Y -453.726,Z 499.994,A 0.000,B 0.000,C 90.000,E1 214.898} C_DIS
LIN {X -0.142,Y -449.318,Z 499.981,A 0.000,B 0.000,C 90.000,E1 212.673} C_DIS
LIN {X -0.141,Y -446.318,Z 499.972,A 0.000,B 0.000,C 90.000,E1 211.052} C_DIS
LIN {X -0.042,Y -443.322,Z 499.963,A 0.000,B 0.000,C 90.000,E1 209.411} C_DIS
LIN {X -0.163,Y -439.815,Z 499.953,A 0.000,B 0.000,C 90.000,E1 207.462} C_DIS
LIN {X -0.001,Y -436.874,Z 499.943,A 0.000,B 0.000,C 90.000,E1 205.796} C_DIS
LIN {X -0.084,Y -433.397,Z 499.932,A 0.000,B 0.000,C 90.000,E1 203.823} C_DIS
LIN {X -0.203,Y -430.038,Z 499.921,A 0.000,B 0.000,C 90.000,E1 201.844} C_DIS
LIN {X 0.196,Y -427.349,Z 499.912,A 0.000,B 0.000,C 90.000,E1 200.120} C_DIS
LIN {X 0.019,Y -423.390,Z 499.897,A 0.000,B 0.000,C 90.000,E1 197.457} C_DIS
LIN {X -0.126,Y -419.810,Z 499.882,A 0.000,B 0.000,C 90.000,E1 194.773} C_DIS
LIN {X 0.018,Y -417.347,Z 499.871,A 0.000,B 0.000,C 90.000,E1 192.715} C_DIS
LIN {X 0.148,Y -414.662,Z 499.857,A 0.000,B 0.000,C 90.000,E1 190.310} C_DIS
LIN {X 0.001,Y -412.444,Z 499.846,A 0.000,B 0.000,C 90.000,E1 188.276} C_DIS
LIN {X 0.095,Y -410.444,Z 499.835,A 0.000,B 0.000,C 90.000,E1 186.201} C_DIS
LIN {X 0.125,Y -408.711,Z 499.825,A 0.000,B 0.000,C 90.000,E1 184.473} C_DIS
LIN {X 0.018,Y -406.107,Z 499.808,A 0.000,B 0.000,C 90.000,E1 181.375} C_DIS
LIN {X -0.153,Y -404.576,Z 499.794,A 0.000,B 0.000,C 90.000,E1 178.969} C_DIS
LIN {X -0.077,Y -402.894,Z 499.771,A 0.000,B 0.000,C 90.000,E1 174.780} C_DIS
LIN {X 0.191,Y -402.566,Z 499.755,A 0.000,B 0.000,C 90.000,E1 171.951} C_DIS
LIN {X 0.173,Y -402.789,Z 499.740,A 0.000,B 0.000,C 90.000,E1 169.162} C_DIS
LIN {X -0.081,Y -403.455,Z 499.724,A 0.000,B 0.000,C 90.000,E1 166.408} C_DIS
LIN {X -0.035,Y -404.702,Z 499.707,A 0.000,B 0.000,C 90.000,E1 163.268} C_DIS
LIN {X 0.015,Y -406.526,Z 499.690,A 0.000,B 0.000,C 90.000,E1 160.134} C_DIS
LIN {X 0.055,Y -408.582,Z 499.674,A 0.000,B 0.000,C 90.000,E1 157.358} C_DIS
LIN {X -0.166,Y -410.662,Z 499.661,A 0.000,B 0.000,C 90.000,E1 154.973} C_DIS
LIN {X 0.100,Y -412.582,Z 499.649,A 0.000,B 0.000,C 90.000,E1 152.871} C_DIS
LIN {X -0.131,Y -414.404,Z 499.638,A 0.000,B 0.000,C 90.000,E1 150.845} C_DIS
LIN {X -0.003,Y -415.546,Z 499.630,A 0.000,B 0.000,C 90.000,E1 149.459} C_DIS
LIN {X 0.085,Y -416.981,Z 499.621,A 0.000,B 0.000,C 90.000,E1 147.740} C_DIS
LIN {X 0.108,Y -418.056,Z 499.613,A 0.000,B 0.000,C 90.000,E1 146.373} C_DIS
LIN {X -0.007,Y -419.353,Z 499.604,A 0.000,B 0.000,C 90.000,E1 144.689} C_DIS
LIN {X 0.106,Y -420.869,Z 499.593,A 0.000,B 0.000,C 90.000,E1 142.637} C_DIS
LIN {X -0.156,Y -422.309,Z 499.581,A 0.000,B 0.000,C 90.000,E1 140.642} C_DIS
LIN {X 0.100,Y -423.187,Z 499.574,A 0.000,B 0.000,C 90.000,E1 139.256} C_DIS
LIN {X 0.005,Y -423.962,Z 499.566,A 0.000,B 0.000,C 90.000,E1 137.919} C_DIS
LIN {X 0.122,Y -424.304,Z 499.563,A 0.000,B 0.000,C 90.000,E1 137.229} C_DIS
LIN {X 0.052,Y -424.749,Z 499.555,A 0.000,B 0.000,C 90.000,E1 135.891} C_DIS
LIN {X -0.226,Y -425.055,Z 499.549,A 0.000,B 0.000,C 90.000,E1 134.919} C_DIS
LIN {X 0.009,Y -425.195,Z 499.542,A 0.000,B 0.000,C 90.000,E1 133.542} C_DIS
LIN {X 0.040,Y -425.031,Z 499.536,A 0.000,B 0.000,C 90.000,E1 132.528} C_DIS
LIN {X -0.028,Y -424.404,Z 499.529,A 0.000,B 0.000,C 90.000,E1 131.191} C_DIS
LIN {X 0.035,Y -423.773,Z 499.523,A 0.000,B 0.000,C 90.000,E1 130.172} C_DIS
LIN {X 0.204,Y -422.180,Z 499.514,A 0.000,B 0.000,C 90.000,E1 128.463} C_DIS
LIN {X -0.133,Y -420.833,Z 499.506,A 0.000,B 0.000,C 90.000,E1 127.156} C_DIS
LIN {X -0.154,Y -419.372,Z 499.499,A 0.000,B 0.000,C 90.000,E1 125.804} C_DIS
LIN {X 0.071,Y -418.224,Z 499.494,A 0.000,B 0.000,C 90.000,E1 124.818} C_DIS
LIN {X 0.032,Y -418.218,Z 499.493,A 0.000,B 0.000,C 90.000,E1 124.818} C_DIS
LIN {X -0.040,Y -427.427,Z 499.474,A 0.000,B 0.000,C 90.000,E1 121.386} C_DIS
LIN {X -0.068,Y -430.497,Z 499.469,A 0.000,B 0.000,C 90.000,E1 120.384} C_DIS
LIN {X 0.112,Y -433.620,Z 499.461,A 0.000,B 0.000,C 90.000,E1 119.027} C_DIS
LIN {X -0.015,Y -443.336,Z 499.441,A 0.000,B 0.000,C 90.000,E1 115.412} C_DIS
LIN {X 0.025,Y -444.324,Z 499.439,A 0.000,B 0.000,C 90.000,E1 115.079} C_DIS
LIN {X -0.123,Y -445.159,Z 499.438,A 0.000,B 0.000,C 90.000,E1 114.771} C_DIS
LIN {X -0.016,Y -454.343,Z 499.416,A 0.000,B 0.000,C 90.000,E1 110.865} C_DIS
LIN {X 0.105,Y -457.012,Z 499.411,A 0.000,B 0.000,C 90.000,E1 109.885} C_DIS
LIN {X -0.087,Y -458.264,Z 499.407,A 0.000,B 0.000,C 90.000,E1 109.268} C_DIS
LIN {X -0.119,Y -462.630,Z 499.395,A 0.000,B 0.000,C 90.000,E1 107.094} C_DIS
LIN {X -0.160,Y -462.773,Z 499.395,A 0.000,B 0.000,C 90.000,E1 107.094} C_DIS
LIN {X -0.032,Y -476.234,Z 499.393,A 0.000,B 0.000,C 90.000,E1 106.804} C_DIS
LIN {X -0.219,Y -490.098,Z 499.392,A 0.000,B 0.000,C 90.000,E1 106.496} C_DIS
LIN {X -0.124,Y -507.688,Z 499.389,A 0.000,B 0.000,C 90.000,E1 106.024} C_DIS
LIN {X 0.042,Y -521.227,Z 499.387,A 0.000,B 0.000,C 90.000,E1 105.607} C_DIS
LIN {X -0.163,Y -531.695,Z 499.385,A 0.000,B 0.000,C 90.000,E1 105.300} C_DIS
LIN {X -0.193,Y -541.872,Z 499.383,A 0.000,B 0.000,C 90.000,E1 104.954} C_DIS
LIN {X 0.154,Y -548.533,Z 499.382,A 0.000,B 0.000,C 90.000,E1 104.662} C_DIS
LIN {X -0.130,Y -554.937,Z 499.380,A 0.000,B 0.000,C 90.000,E1 104.411} C_DIS
LIN {X 0.264,Y -561.369,Z 499.378,A 0.000,B 0.000,C 90.000,E1 104.064} C_DIS
LIN {X -0.022,Y -567.441,Z 499.377,A 0.000,B 0.000,C 90.000,E1 103.772} C_DIS
LIN {X 0.152,Y -575.101,Z 499.374,A 0.000,B 0.000,C 90.000,E1 103.300} C_DIS
LIN {X 0.048,Y -578.231,Z 499.373,A 0.000,B 0.000,C 90.000,E1 103.119} C_DIS
LIN {X -0.004,Y -584.071,Z 499.371,A 0.000,B 0.000,C 90.000,E1 102.715} C_DIS
LIN {X -0.129,Y -591.160,Z 499.368,A 0.000,B 0.000,C 90.000,E1 102.175} C_DIS
LIN {X -0.095,Y -595.396,Z 499.366,A 0.000,B 0.000,C 90.000,E1 101.827} C_DIS
LIN {X -0.263,Y -602.035,Z 499.362,A 0.000,B 0.000,C 90.000,E1 101.243} C_DIS
LIN {X 0.061,Y -607.213,Z 499.360,A 0.000,B 0.000,C 90.000,E1 100.715} C_DIS
LIN {X 0.218,Y -613.216,Z 499.356,A 0.000,B 0.000,C 90.000,E1 100.074} C_DIS
LIN {X -0.122,Y -619.638,Z 499.352,A 0.000,B 0.000,C 90.000,E1 99.378} C_DIS
LIN {X 0.068,Y -625.670,Z 499.348,A 0.000,B 0.000,C 90.000,E1 98.624} C_DIS
LIN {X -0.202,Y -632.043,Z 499.343,A 0.000,B 0.000,C 90.000,E1 97.757} C_DIS
LIN {X -0.067,Y -636.749,Z 499.339,A 0.000,B 0.000,C 90.000,E1 97.004} C_DIS
LIN {X 0.101,Y -639.782,Z 499.336,A 0.000,B 0.000,C 90.000,E1 96.486} C_DIS
LIN {X 0.045,Y -643.747,Z 499.332,A 0.000,B 0.000,C 90.000,E1 95.739} C_DIS
LIN {X -0.143,Y -648.667,Z 499.326,A 0.000,B 0.000,C 90.000,E1 94.759} C_DIS
LIN {X -0.115,Y -651.996,Z 499.322,A 0.000,B 0.000,C 90.000,E1 94.012} C_DIS
LIN {X 0.111,Y -654.037,Z 499.320,A 0.000,B 0.000,C 90.000,E1 93.498} C_DIS
LIN {X 0.193,Y -656.624,Z 499.315,A 0.000,B 0.000,C 90.000,E1 92.751} C_DIS
LIN {X -0.196,Y -658.123,Z 499.313,A 0.000,B 0.000,C 90.000,E1 92.293} C_DIS
LIN {X 0.106,Y -659.321,Z 499.310,A 0.000,B 0.000,C 90.000,E1 91.776} C_DIS
LIN {X -0.266,Y -660.236,Z 499.307,A 0.000,B 0.000,C 90.000,E1 91.318} C_DIS
LIN {X -0.149,Y -661.151,Z 499.303,A 0.000,B 0.000,C 90.000,E1 90.573} C_DIS
LIN {X 0.156,Y -661.540,Z 499.300,A 0.000,B 0.000,C 90.000,E1 90.057} C_DIS
LIN {X -0.196,Y -661.559,Z 499.298,A 0.000,B 0.000,C 90.000,E1 89.599} C_DIS
LIN {X -0.065,Y -661.129,Z 499.294,A 0.000,B 0.000,C 90.000,E1 88.854} C_DIS
LIN {X 0.238,Y -660.628,Z 499.291,A 0.000,B 0.000,C 90.000,E1 88.339} C_DIS
LIN {X -0.099,Y -659.926,Z 499.288,A 0.000,B 0.000,C 90.000,E1 87.879} C_DIS
LIN {X 0.010,Y -658.399,Z 499.284,A 0.000,B 0.000,C 90.000,E1 87.135} C_DIS
LIN {X 0.325,Y -657.142,Z 499.281,A 0.000,B 0.000,C 90.000,E1 86.617} C_DIS
LIN {X -0.062,Y -655.677,Z 499.279,A 0.000,B 0.000,C 90.000,E1 86.159} C_DIS
LIN {X 0.036,Y -653.089,Z 499.275,A 0.000,B 0.000,C 90.000,E1 85.412} C_DIS
LIN {X 0.106,Y -650.017,Z 499.270,A 0.000,B 0.000,C 90.000,E1 84.666} C_DIS
LIN {X 0.257,Y -647.128,Z 499.267,A 0.000,B 0.000,C 90.000,E1 84.033} C_DIS
LIN {X -0.189,Y -643.935,Z 499.264,A 0.000,B 0.000,C 90.000,E1 83.451} C_DIS
LIN {X -0.090,Y -640.439,Z 499.260,A 0.000,B 0.000,C 90.000,E1 82.818} C_DIS
LIN {X -0.210,Y -634.964,Z 499.255,A 0.000,B 0.000,C 90.000,E1 81.951} C_DIS
LIN {X -0.195,Y -628.980,Z 499.250,A 0.000,B 0.000,C 90.000,E1 81.084} C_DIS
LIN {X -0.136,Y -624.242,Z 499.247,A 0.000,B 0.000,C 90.000,E1 80.443} C_DIS
LIN {X -0.012,Y -618.274,Z 499.243,A 0.000,B 0.000,C 90.000,E1 79.690} C_DIS
LIN {X -0.047,Y -612.655,Z 499.239,A 0.000,B 0.000,C 90.000,E1 79.050} C_DIS
LIN {X -0.014,Y -606.657,Z 499.236,A 0.000,B 0.000,C 90.000,E1 78.409} C_DIS
LIN {X -0.235,Y -602.962,Z 499.234,A 0.000,B 0.000,C 90.000,E1 78.049} C_DIS
LIN {X 0.083,Y -596.153,Z 499.230,A 0.000,B 0.000,C 90.000,E1 77.409} C_DIS
LIN {X 0.175,Y -588.932,Z 499.227,A 0.000,B 0.000,C 90.000,E1 76.825} C_DIS
LIN {X -0.131,Y -584.511,Z 499.225,A 0.000,B 0.000,C 90.000,E1 76.520} C_DIS
LIN {X 0.176,Y -579.928,Z 499.223,A 0.000,B 0.000,C 90.000,E1 76.172} C_DIS
LIN {X -0.187,Y -573.496,Z 499.221,A 0.000,B 0.000,C 90.000,E1 75.811} C_DIS
LIN {X -0.018,Y -568.470,Z 499.220,A 0.000,B 0.000,C 90.000,E1 75.519} C_DIS
LIN {X 0.141,Y -561.232,Z 499.218,A 0.000,B 0.000,C 90.000,E1 75.172} C_DIS
LIN {X -0.196,Y -555.844,Z 499.217,A 0.000,B 0.000,C 90.000,E1 74.991} C_DIS
LIN {X -0.267,Y -548.207,Z 499.215,A 0.000,B 0.000,C 90.000,E1 74.755} C_DIS
LIN {X 0.023,Y -542.208,Z 499.214,A 0.000,B 0.000,C 90.000,E1 74.574} C_DIS
LIN {X 0.075,Y -536.611,Z 499.214,A 0.000,B 0.000,C 90.000,E1 74.448} C_DIS
LIN {X -0.137,Y -528.581,Z 499.213,A 0.000,B 0.000,C 90.000,E1 74.338} C_DIS
LIN {X -0.183,Y -524.059,Z 499.213,A 0.000,B 0.000,C 90.000,E1 74.283} C_DIS
LIN {X 0.003,Y -510.820,Z 499.212,A 0.000,B 0.000,C 90.000,E1 74.157} C_DIS
LIN {X -0.280,Y -494.359,Z 499.212,A 0.000,B 0.000,C 90.000,E1 74.102} C_DIS
LIN {X 0.156,Y -476.386,Z 499.212,A 0.000,B 0.000,C 90.000,E1 74.047} C_DIS
LIN {X 0.061,Y -474.136,Z 499.200,A 0.000,B 0.000,C 90.000,E1 72.054} C_DIS
LIN {X -0.072,Y -465.608,Z 499.172,A 0.000,B 0.000,C 90.000,E1 67.050} C_DIS
LIN {X -0.193,Y -456.604,Z 499.148,A 0.000,B 0.000,C 90.000,E1 62.615} C_DIS
LIN {X -0.194,Y -455.562,Z 499.144,A 0.000,B 0.000,C 90.000,E1 61.975} C_DIS
LIN {X 0.009,Y -449.993,Z 499.131,A 0.000,B 0.000,C 90.000,E1 59.587} C_DIS
LIN {X -0.031,Y -449.989,Z 499.131,A 0.000,B 0.000,C 90.000,E1 59.587} C_DIS
LIN {X -0.123,Y -454.704,Z 499.125,A 0.000,B 0.000,C 90.000,E1 58.584} C_DIS
LIN {X 0.193,Y -458.942,Z 499.120,A 0.000,B 0.000,C 90.000,E1 57.582} C_DIS
LIN {X 0.044,Y -464.342,Z 499.112,A 0.000,B 0.000,C 90.000,E1 56.167} C_DIS
LIN {X -0.073,Y -466.360,Z 499.109,A 0.000,B 0.000,C 90.000,E1 55.548} C_DIS
LIN {X -0.143,Y -469.010,Z 499.103,A 0.000,B 0.000,C 90.000,E1 54.609} C_DIS
LIN {X 0.206,Y -471.107,Z 499.098,A 0.000,B 0.000,C 90.000,E1 53.623} C_DIS
LIN {X 0.137,Y -472.392,Z 499.095,A 0.000,B 0.000,C 90.000,E1 53.004} C_DIS
LIN {X 0.007,Y -474.763,Z 499.086,A 0.000,B 0.000,C 90.000,E1 51.457} C_DIS
LIN {X 0.040,Y -475.887,Z 499.081,A 0.000,B 0.000,C 90.000,E1 50.517} C_DIS
LIN {X -0.183,Y -477.025,Z 499.074,A 0.000,B 0.000,C 90.000,E1 49.299} C_DIS
LIN {X 0.178,Y -477.772,Z 499.069,A 0.000,B 0.000,C 90.000,E1 48.324} C_DIS
LIN {X 0.191,Y -478.355,Z 499.063,A 0.000,B 0.000,C 90.000,E1 47.391} C_DIS
LIN {X 0.209,Y -478.811,Z 499.058,A 0.000,B 0.000,C 90.000,E1 46.458} C_DIS
LIN {X 0.126,Y -479.252,Z 499.050,A 0.000,B 0.000,C 90.000,E1 44.919} C_DIS
LIN {X -0.070,Y -479.391,Z 499.043,A 0.000,B 0.000,C 90.000,E1 43.704} C_DIS
LIN {X 0.078,Y -479.228,Z 499.036,A 0.000,B 0.000,C 90.000,E1 42.447} C_DIS
LIN {X -0.097,Y -478.806,Z 499.029,A 0.000,B 0.000,C 90.000,E1 41.229} C_DIS
LIN {X -0.006,Y -477.929,Z 499.019,A 0.000,B 0.000,C 90.000,E1 39.358} C_DIS
LIN {X 0.164,Y -477.277,Z 499.012,A 0.000,B 0.000,C 90.000,E1 38.096} C_DIS
LIN {X 0.027,Y -476.583,Z 499.005,A 0.000,B 0.000,C 90.000,E1 36.870} C_DIS
LIN {X 0.057,Y -475.609,Z 498.996,A 0.000,B 0.000,C 90.000,E1 35.311} C_DIS
LIN {X -0.206,Y -474.380,Z 498.988,A 0.000,B 0.000,C 90.000,E1 33.785} C_DIS
LIN {X -0.097,Y -473.106,Z 498.979,A 0.000,B 0.000,C 90.000,E1 32.212} C_DIS
LIN {X 0.209,Y -472.022,Z 498.972,A 0.000,B 0.000,C 90.000,E1 30.924} C_DIS
LIN {X 0.252,Y -470.820,Z 498.965,A 0.000,B 0.000,C 90.000,E1 29.667} C_DIS
LIN {X -0.263,Y -469.029,Z 498.955,A 0.000,B 0.000,C 90.000,E1 27.847} C_DIS
LIN {X 0.105,Y -466.871,Z 498.941,A 0.000,B 0.000,C 90.000,E1 25.283} C_DIS
LIN {X -0.057,Y -464.776,Z 498.925,A 0.000,B 0.000,C 90.000,E1 22.461} C_DIS
LIN {X -0.148,Y -463.310,Z 498.911,A 0.000,B 0.000,C 90.000,E1 19.939} C_DIS
LIN {X 0.139,Y -462.383,Z 498.900,A 0.000,B 0.000,C 90.000,E1 18.000} C_DIS
LIN {X -0.047,Y -461.397,Z 498.886,A 0.000,B 0.000,C 90.000,E1 15.481} C_DIS
LIN {X 0.167,Y -460.663,Z 498.870,A 0.000,B 0.000,C 90.000,E1 12.591} C_DIS
LIN {X -0.082,Y -460.506,Z 498.856,A 0.000,B 0.000,C 90.000,E1 10.074} C_DIS
LIN {X 0.131,Y -460.893,Z 498.840,A 0.000,B 0.000,C 90.000,E1 7.182} C_DIS
LIN {X -0.221,Y -462.199,Z 498.821,A 0.000,B 0.000,C 90.000,E1 3.726} C_DIS
LIN {X 0.111,Y -463.797,Z 498.806,A 0.000,B 0.000,C 90.000,E1 1.146} C_DIS
LIN {X -0.106,Y -466.982,Z 498.787,A 0.000,B 0.000,C 90.000,E1 357.593} C_DIS
LIN {X 0.127,Y -468.698,Z 498.778,A 0.000,B 0.000,C 90.000,E1 355.988} C_DIS
LIN {X -0.242,Y -470.985,Z 498.767,A 0.000,B 0.000,C 90.000,E1 354.147} C_DIS
LIN {X 0.139,Y -472.980,Z 498.759,A 0.000,B 0.000,C 90.000,E1 352.534} C_DIS
LIN {X -0.180,Y -475.896,Z 498.747,A 0.000,B 0.000,C 90.000,E1 350.387} C_DIS
LIN {X -0.163,Y -480.291,Z 498.731,A 0.000,B 0.000,C 90.000,E1 347.589} C_DIS
LIN {X 0.142,Y -483.691,Z 498.721,A 0.000,B 0.000,C 90.000,E1 345.700} C_DIS
LIN {X -0.065,Y -488.629,Z 498.707,A 0.000,B 0.000,C 90.000,E1 343.268} C_DIS
LIN {X -0.231,Y -492.506,Z 498.697,A 0.000,B 0.000,C 90.000,E1 341.456} C_DIS
LIN {X -0.138,Y -496.565,Z 498.687,A 0.000,B 0.000,C 90.000,E1 339.625} C_DIS
LIN {X 0.044,Y -500.515,Z 498.677,A 0.000,B 0.000,C 90.000,E1 337.794} C_DIS
LIN {X -0.055,Y -503.703,Z 498.668,A 0.000,B 0.000,C 90.000,E1 336.305} C_DIS
LIN {X 0.022,Y -506.207,Z 498.662,A 0.000,B 0.000,C 90.000,E1 335.101} C_DIS
LIN {X 0.194,Y -510.463,Z 498.650,A 0.000,B 0.000,C 90.000,E1 332.999} C_DIS
LIN {X -0.096,Y -514.115,Z 498.640,A 0.000,B 0.000,C 90.000,E1 331.257} C_DIS
LIN {X -0.084,Y -516.671,Z 498.634,A 0.000,B 0.000,C 90.000,E1 330.078} C_DIS
LIN {X 0.198,Y -521.179,Z 498.622,A 0.000,B 0.000,C 90.000,E1 327.995} C_DIS
LIN {X 0.155,Y -525.732,Z 498.611,A 0.000,B 0.000,C 90.000,E1 325.960} C_DIS
LIN {X -0.024,Y -529.718,Z 498.601,A 0.000,B 0.000,C 90.000,E1 324.242} C_DIS
LIN {X 0.325,Y -533.735,Z 498.592,A 0.000,B 0.000,C 90.000,E1 322.477} C_DIS
LIN {X -0.101,Y -537.000,Z 498.584,A 0.000,B 0.000,C 90.000,E1 321.090} C_DIS
LIN {X -0.116,Y -540.891,Z 498.574,A 0.000,B 0.000,C 90.000,E1 319.380} C_DIS
LIN {X -0.101,Y -544.804,Z 498.565,A 0.000,B 0.000,C 90.000,E1 317.676} C_DIS
LIN {X -0.002,Y -548.584,Z 498.555,A 0.000,B 0.000,C 90.000,E1 315.972} C_DIS
LIN {X -0.197,Y -552.814,Z 498.545,A 0.000,B 0.000,C 90.000,E1 314.028} C_DIS
LIN {X 0.103,Y -557.008,Z 498.534,A 0.000,B 0.000,C 90.000,E1 312.043} C_DIS
LIN {X 0.090,Y -560.587,Z 498.524,A 0.000,B 0.000,C 90.000,E1 310.378} C_DIS
LIN {X -0.207,Y -564.096,Z 498.515,A 0.000,B 0.000,C 90.000,E1 308.749} C_DIS
LIN {X 0.252,Y -568.868,Z 498.503,A 0.000,B 0.000,C 90.000,E1 306.503} C_DIS
LIN {X 0.034,Y -573.099,Z 498.492,A 0.000,B 0.000,C 90.000,E1 304.612} C_DIS
LIN {X 0.246,Y -576.734,Z 498.483,A 0.000,B 0.000,C 90.000,E1 302.959} C_DIS
LIN {X 0.069,Y -579.737,Z 498.476,A 0.000,B 0.000,C 90.000,E1 301.623} C_DIS
LIN {X 0.089,Y -581.985,Z 498.470,A 0.000,B 0.000,C 90.000,E1 300.541} C_DIS
LIN {X 0.000,Y -584.640,Z 498.462,A 0.000,B 0.000,C 90.000,E1 299.205} C_DIS
LIN {X -0.219,Y -586.586,Z 498.456,A 0.000,B 0.000,C 90.000,E1 298.153} C_DIS
LIN {X 0.103,Y -588.324,Z 498.450,A 0.000,B 0.000,C 90.000,E1 297.052} C_DIS
LIN {X 0.295,Y -589.423,Z 498.446,A 0.000,B 0.000,C 90.000,E1 296.232} C_DIS
LIN {X 0.294,Y -591.027,Z 498.439,A 0.000,B 0.000,C 90.000,E1 294.899} C_DIS
LIN {X -0.123,Y -592.018,Z 498.433,A 0.000,B 0.000,C 90.000,E1 293.875} C_DIS
LIN {X 0.213,Y -593.018,Z 498.425,A 0.000,B 0.000,C 90.000,E1 292.514} C_DIS
LIN {X 0.251,Y -594.070,Z 498.416,A 0.000,B 0.000,C 90.000,E1 290.918} C_DIS
LIN {X -0.142,Y -594.762,Z 498.409,A 0.000,B 0.000,C 90.000,E1 289.631} C_DIS
LIN {X 0.290,Y -595.293,Z 498.400,A 0.000,B 0.000,C 90.000,E1 288.000} C_DIS
LIN {X 0.283,Y -595.684,Z 498.393,A 0.000,B 0.000,C 90.000,E1 286.677} C_DIS
LIN {X -0.180,Y -596.050,Z 498.384,A 0.000,B 0.000,C 90.000,E1 285.134} C_DIS
LIN {X -0.048,Y -596.243,Z 498.378,A 0.000,B 0.000,C 90.000,E1 284.064} C_DIS
LIN {X 0.230,Y -596.376,Z 498.371,A 0.000,B 0.000,C 90.000,E1 282.715} C_DIS
LIN {X 0.221,Y -596.439,Z 498.362,A 0.000,B 0.000,C 90.000,E1 281.130} C_DIS
LIN {X -0.198,Y -596.363,Z 498.355,A 0.000,B 0.000,C 90.000,E1 279.849} C_DIS
LIN {X -0.033,Y -596.133,Z 498.347,A 0.000,B 0.000,C 90.000,E1 278.511} C_DIS
LIN {X 0.038,Y -595.753,Z 498.340,A 0.000,B 0.000,C 90.000,E1 277.182} C_DIS
LIN {X -0.175,Y -595.333,Z 498.334,A 0.000,B 0.000,C 90.000,E1 276.144} C_DIS
LIN {X 0.083,Y -594.387,Z 498.325,A 0.000,B 0.000,C 90.000,E1 274.531} C_DIS
LIN {X 0.176,Y -593.805,Z 498.321,A 0.000,B 0.000,C 90.000,E1 273.726} C_DIS
LIN {X -0.115,Y -592.920,Z 498.315,A 0.000,B 0.000,C 90.000,E1 272.694} C_DIS
LIN {X -0.211,Y -591.488,Z 498.308,A 0.000,B 0.000,C 90.000,E1 271.375} C_DIS
LIN {X 0.040,Y -590.197,Z 498.302,A 0.000,B 0.000,C 90.000,E1 270.286} C_DIS
LIN {X -0.114,Y -588.436,Z 498.294,A 0.000,B 0.000,C 90.000,E1 268.969} C_DIS
LIN {X -0.093,Y -586.209,Z 498.285,A 0.000,B 0.000,C 90.000,E1 267.364} C_DIS
LIN {X -0.085,Y -583.903,Z 498.276,A 0.000,B 0.000,C 90.000,E1 265.755} C_DIS
LIN {X 0.288,Y -581.794,Z 498.269,A 0.000,B 0.000,C 90.000,E1 264.375} C_DIS
LIN {X -0.106,Y -578.435,Z 498.258,A 0.000,B 0.000,C 90.000,E1 262.527} C_DIS
LIN {X -0.017,Y -575.097,Z 498.248,A 0.000,B 0.000,C 90.000,E1 260.622} C_DIS
LIN {X -0.127,Y -572.679,Z 498.240,A 0.000,B 0.000,C 90.000,E1 259.275} C_DIS
LIN {X 0.175,Y -570.024,Z 498.233,A 0.000,B 0.000,C 90.000,E1 257.881} C_DIS
LIN {X 0.287,Y -566.684,Z 498.224,A 0.000,B 0.000,C 90.000,E1 256.228} C_DIS
LIN {X -0.134,Y -564.415,Z 498.218,A 0.000,B 0.000,C 90.000,E1 255.172} C_DIS
LIN {X -0.142,Y -561.399,Z 498.210,A 0.000,B 0.000,C 90.000,E1 253.795} C_DIS
LIN {X 0.041,Y -558.810,Z 498.204,A 0.000,B 0.000,C 90.000,E1 252.670} C_DIS
LIN {X -0.185,Y -556.132,Z 498.198,A 0.000,B 0.000,C 90.000,E1 251.583} C_DIS
LIN {X -0.025,Y -554.001,Z 498.193,A 0.000,B 0.000,C 90.000,E1 250.732} C_DIS
LIN {X -0.046,Y -550.295,Z 498.185,A 0.000,B 0.000,C 90.000,E1 249.337} C_DIS
LIN {X 0.246,Y -547.963,Z 498.181,A 0.000,B 0.000,C 90.000,E1 248.465} C_DIS
LIN {X -0.195,Y -544.001,Z 498.173,A 0.000,B 0.000,C 90.000,E1 247.102} C_DIS
LIN {X 0.269,Y -540.614,Z 498.166,A 0.000,B 0.000,C 90.000,E1 245.921} C_DIS
LIN {X -0.089,Y -536.275,Z 498.159,A 0.000,B 0.000,C 90.000,E1 244.537} C_DIS
LIN {X -0.005,Y -532.724,Z 498.152,A 0.000,B 0.000,C 90.000,E1 243.384} C_DIS
LIN {X -0.023,Y -528.203,Z 498.144,A 0.000,B 0.000,C 90.000,E1 241.948} C_DIS
LIN {X -0.035,Y -521.825,Z 498.133,A 0.000,B 0.000,C 90.000,E1 239.921} C_DIS
LIN {X 0.012,Y -517.252,Z 498.125,A 0.000,B 0.000,C 90.000,E1 238.456} C_DIS
LIN {X -0.037,Y -514.446,Z 498.120,A 0.000,B 0.000,C 90.000,E1 237.582} C_DIS
LIN {X 0.048,Y -508.685,Z 498.110,A 0.000,B 0.000,C 90.000,E1 235.801} C_DIS
LIN {X -0.126,Y -502.809,Z 498.100,A 0.000,B 0.000,C 90.000,E1 234.036} C_DIS
LIN {X 0.270,Y -497.089,Z 498.090,A 0.000,B 0.000,C 90.000,E1 232.190} C_DIS
LIN {X -0.245,Y -489.963,Z 498.077,A 0.000,B 0.000,C 90.000,E1 229.828} C_DIS
LIN {X 0.212,Y -484.017,Z 498.065,A 0.000,B 0.000,C 90.000,E1 227.634} C_DIS
LIN {X -0.001,Y -479.059,Z 498.055,A 0.000,B 0.000,C 90.000,E1 225.810} C_DIS
LIN {X 0.113,Y -473.478,Z 498.042,A 0.000,B 0.000,C 90.000,E1 223.623} C_DIS
LIN {X 0.013,Y -468.846,Z 498.032,A 0.000,B 0.000,C 90.000,E1 221.757} C_DIS
LIN {X -0.043,Y -463.051,Z 498.018,A 0.000,B 0.000,C 90.000,E1 219.241} C_DIS
LIN {X 0.115,Y -458.239,Z 498.006,A 0.000,B 0.000,C 90.000,E1 216.996} C_DIS
LIN {X -0.116,Y -454.339,Z 497.995,A 0.000,B 0.000,C 90.000,E1 215.105} C_DIS
LIN {X -0.056,Y -450.531,Z 497.984,A 0.000,B 0.000,C 90.000,E1 213.166} C_DIS
LIN {X 0.049,Y -446.926,Z 497.973,A 0.000,B 0.000,C 90.000,E1 211.209} C_DIS
LIN {X -0.158,Y -443.343,Z 497.963,A 0.000,B 0.000,C 90.000,E1 209.283} C_DIS
LIN {X -0.075,Y -439.830,Z 497.952,A 0.000,B 0.000,C 90.000,E1 207.308} C_DIS
LIN {X -0.114,Y -436.860,Z 497.943,A 0.000,B 0.000,C 90.000,E1 205.668} C_DIS
LIN {X -0.022,Y -433.969,Z 497.933,A 0.000,B 0.000,C 90.000,E1 204.003} C_DIS
LIN {X -0.133,Y -430.596,Z 497.922,A 0.000,B 0.000,C 90.000,E1 202.025} C_DIS
LIN {X 0.081,Y -426.301,Z 497.907,A 0.000,B 0.000,C 90.000,E1 199.322} C_DIS
LIN {X 0.114,Y -423.847,Z 497.898,A 0.000,B 0.000,C 90.000,E1 197.638} C_DIS
LIN {X -0.017,Y -420.213,Z 497.883,A 0.000,B 0.000,C 90.000,E1 194.954} C_DIS
LIN {X -0.175,Y -417.713,Z 497.872,A 0.000,B 0.000,C 90.000,E1 192.939} C_DIS
LIN {X -0.172,Y -415.376,Z 497.860,A 0.000,B 0.000,C 90.000,E1 190.894} C_DIS
LIN {X 0.111,Y -413.117,Z 497.849,A 0.000,B 0.000,C 90.000,E1 188.803} C_DIS
LIN {X -0.100,Y -410.748,Z 497.836,A 0.000,B 0.000,C 90.000,E1 186.429} C_DIS
LIN {X -0.086,Y -408.671,Z 497.824,A 0.000,B 0.000,C 90.000,E1 184.359} C_DIS
LIN {X -0.190,Y -406.119,Z 497.807,A 0.000,B 0.000,C 90.000,E1 181.260} C_DIS
LIN {X 0.046,Y -404.593,Z 497.793,A 0.000,B 0.000,C 90.000,E1 178.797} C_DIS
LIN {X 0.161,Y -403.039,Z 497.772,A 0.000,B 0.000,C 90.000,E1 174.951} C_DIS
LIN {X -0.013,Y -402.695,Z 497.757,A 0.000,B 0.000,C 90.000,E1 172.186} C_DIS
LIN {X -0.038,Y -402.911,Z 497.739,A 0.000,B 0.000,C 90.000,E1 169.050} C_DIS
LIN {X 0.192,Y -403.641,Z 497.724,A 0.000,B 0.000,C 90.000,E1 166.228} C_DIS
LIN {X 0.150,Y -404.757,Z 497.708,A 0.000,B 0.000,C 90.000,E1 163.449} C_DIS
LIN {X -0.181,Y -406.584,Z 497.691,A 0.000,B 0.000,C 90.000,E1 160.369} C_DIS
LIN {X -0.131,Y -408.643,Z 497.675,A 0.000,B 0.000,C 90.000,E1 157.592} C_DIS
LIN {X 0.123,Y -410.436,Z 497.664,A 0.000,B 0.000,C 90.000,E1 155.485} C_DIS
LIN {X 0.123,Y -412.684,Z 497.651,A 0.000,B 0.000,C 90.000,E1 153.076} C_DIS
LIN {X -0.048,Y -414.240,Z 497.641,A 0.000,B 0.000,C 90.000,E1 151.385} C_DIS
LIN {X 0.073,Y -415.482,Z 497.633,A 0.000,B 0.000,C 90.000,E1 149.999} C_DIS
LIN {X 0.107,Y -417.221,Z 497.622,A 0.000,B 0.000,C 90.000,E1 147.946} C_DIS
LIN {X -0.263,Y -418.597,Z 497.613,A 0.000,B 0.000,C 90.000,E1 146.294} C_DIS
LIN {X -0.023,Y -419.928,Z 497.603,A 0.000,B 0.000,C 90.000,E1 144.562} C_DIS
LIN {X -0.236,Y -421.545,Z 497.592,A 0.000,B 0.000,C 90.000,E1 142.557} C_DIS
LIN {X -0.154,Y -423.037,Z 497.581,A 0.000,B 0.000,C 90.000,E1 140.517} C_DIS
LIN {X 0.064,Y -423.969,Z 497.573,A 0.000,B 0.000,C 90.000,E1 139.138} C_DIS
LIN {X 0.021,Y -424.770,Z 497.566,A 0.000,B 0.000,C 90.000,E1 137.796} C_DIS
LIN {X -0.046,Y -425.390,Z 497.558,A 0.000,B 0.000,C 90.000,E1 136.458} C_DIS
LIN {X 0.195,Y -425.891,Z 497.551,A 0.000,B 0.000,C 90.000,E1 135.081} C_DIS
LIN {X 0.063,Y -426.103,Z 497.541,A 0.000,B 0.000,C 90.000,E1 133.419} C_DIS
LIN {X -0.204,Y -425.933,Z 497.536,A 0.000,B 0.000,C 90.000,E1 132.447} C_DIS
LIN {X 0.061,Y -425.319,Z 497.528,A 0.000,B 0.000,C 90.000,E1 131.067} C_DIS
LIN {X 0.189,Y -424.924,Z 497.525,A 0.000,B 0.000,C 90.000,E1 130.378} C_DIS
LIN {X 0.156,Y -423.676,Z 497.517,A 0.000,B 0.000,C 90.000,E1 129.036} C_DIS
LIN {X -0.160,Y -422.312,Z 497.510,A 0.000,B 0.000,C 90.000,E1 127.729} C_DIS
LIN {X -0.158,Y -420.836,Z 497.502,A 0.000,B 0.000,C 90.000,E1 126.377} C_DIS
LIN {X 0.206,Y -419.643,Z 497.496,A 0.000,B 0.000,C 90.000,E1 125.311} C_DIS
LIN {X 0.087,Y -418.713,Z 497.492,A 0.000,B 0.000,C 90.000,E1 124.612} C_DIS
LIN {X 0.048,Y -418.711,Z 497.492,A 0.000,B 0.000,C 90.000,E1 124.612} C_DIS
LIN {X 0.142,Y -428.740,Z 497.472,A 0.000,B 0.000,C 90.000,E1 120.924} C_DIS
LIN {X 0.132,Y -430.798,Z 497.468,A 0.000,B 0.000,C 90.000,E1 120.256} C_DIS
LIN {X 0.092,Y -440.761,Z 497.446,A 0.000,B 0.000,C 90.000,E1 116.283} C_DIS
LIN {X 0.062,Y -444.626,Z 497.439,A 0.000,B 0.000,C 90.000,E1 114.975} C_DIS
LIN {X 0.118,Y -455.484,Z 497.414,A 0.000,B 0.000,C 90.000,E1 110.429} C_DIS
LIN {X -0.083,Y -457.270,Z 497.410,A 0.000,B 0.000,C 90.000,E1 109.812} C_DIS
LIN {X -0.014,Y -463.523,Z 497.393,A 0.000,B 0.000,C 90.000,E1 106.677} C_DIS
LIN {X -0.054,Y -463.572,Z 497.393,A 0.000,B 0.000,C 90.000,E1 106.677} C_DIS
LIN {X 0.133,Y -477.561,Z 497.391,A 0.000,B 0.000,C 90.000,E1 106.386} C_DIS
LIN {X 0.109,Y -491.499,Z 497.389,A 0.000,B 0.000,C 90.000,E1 106.079} C_DIS
LIN {X 0.175,Y -505.829,Z 497.387,A 0.000,B 0.000,C 90.000,E1 105.717} C_DIS
LIN {X -0.135,Y -519.557,Z 497.385,A 0.000,B 0.000,C 90.000,E1 105.371} C_DIS
LIN {X -0.200,Y -529.885,Z 497.384,A 0.000,B 0.000,C 90.000,E1 105.064} C_DIS
LIN {X -0.142,Y -540.174,Z 497.382,A 0.000,B 0.000,C 90.000,E1 104.717} C_DIS
LIN {X -0.207,Y -546.827,Z 497.380,A 0.000,B 0.000,C 90.000,E1 104.481} C_DIS
LIN {X 0.030,Y -553.347,Z 497.379,A 0.000,B 0.000,C 90.000,E1 104.189} C_DIS
LIN {X 0.112,Y -559.914,Z 497.377,A 0.000,B 0.000,C 90.000,E1 103.883} C_DIS
LIN {X -0.119,Y -566.405,Z 497.375,A 0.000,B 0.000,C 90.000,E1 103.592} C_DIS
LIN {X -0.181,Y -575.631,Z 497.373,A 0.000,B 0.000,C 90.000,E1 103.063} C_DIS
LIN {X -0.135,Y -580.104,Z 497.371,A 0.000,B 0.000,C 90.000,E1 102.771} C_DIS
LIN {X -0.260,Y -584.465,Z 497.369,A 0.000,B 0.000,C 90.000,E1 102.479} C_DIS
LIN {X -0.073,Y -587.314,Z 497.368,A 0.000,B 0.000,C 90.000,E1 102.243} C_DIS
LIN {X 0.112,Y -590.350,Z 497.367,A 0.000,B 0.000,C 90.000,E1 102.007} C_DIS
LIN {X 0.273,Y -597.361,Z 497.364,A 0.000,B 0.000,C 90.000,E1 101.422} C_DIS
LIN {X 0.155,Y -601.480,Z 497.362,A 0.000,B 0.000,C 90.000,E1 101.074} C_DIS
LIN {X 0.119,Y -603.986,Z 497.360,A 0.000,B 0.000,C 90.000,E1 100.838} C_DIS
LIN {X 0.031,Y -606.165,Z 497.359,A 0.000,B 0.000,C 90.000,E1 100.658} C_DIS
LIN {X 0.177,Y -613.472,Z 497.355,A 0.000,B 0.000,C 90.000,E1 99.905} C_DIS
LIN {X 0.163,Y -618.805,Z 497.352,A 0.000,B 0.000,C 90.000,E1 99.321} C_DIS
LIN {X -0.247,Y -625.000,Z 497.348,A 0.000,B 0.000,C 90.000,E1 98.624} C_DIS
LIN {X -0.009,Y -627.969,Z 497.346,A 0.000,B 0.000,C 90.000,E1 98.219} C_DIS
LIN {X 0.100,Y -631.679,Z 497.343,A 0.000,B 0.000,C 90.000,E1 97.701} C_DIS
LIN {X 0.039,Y -636.551,Z 497.339,A 0.000,B 0.000,C 90.000,E1 96.947} C_DIS
LIN {X 0.209,Y -639.616,Z 497.336,A 0.000,B 0.000,C 90.000,E1 96.429} C_DIS
LIN {X 0.152,Y -643.613,Z 497.332,A 0.000,B 0.000,C 90.000,E1 95.682} C_DIS
LIN {X -0.035,Y -648.551,Z 497.326,A 0.000,B 0.000,C 90.000,E1 94.702} C_DIS
LIN {X -0.007,Y -651.876,Z 497.322,A 0.000,B 0.000,C 90.000,E1 93.955} C_DIS
LIN {X 0.219,Y -653.903,Z 497.319,A 0.000,B 0.000,C 90.000,E1 93.440} C_DIS
LIN {X -0.154,Y -655.691,Z 497.317,A 0.000,B 0.000,C 90.000,E1 92.980} C_DIS
LIN {X 0.104,Y -657.263,Z 497.314,A 0.000,B 0.000,C 90.000,E1 92.465} C_DIS
LIN {X 0.211,Y -659.092,Z 497.310,A 0.000,B 0.000,C 90.000,E1 91.718} C_DIS
LIN {X -0.161,Y -660.010,Z 497.307,A 0.000,B 0.000,C 90.000,E1 91.260} C_DIS
LIN {X -0.046,Y -660.846,Z 497.303,A 0.000,B 0.000,C 90.000,E1 90.516} C_DIS
LIN {X 0.258,Y -661.198,Z 497.300,A 0.000,B 0.000,C 90.000,E1 90.000} C_DIS
LIN {X -0.097,Y -661.219,Z 497.297,A 0.000,B 0.000,C 90.000,E1 89.542} C_DIS
LIN {X 0.030,Y -660.724,Z 497.293,A 0.000,B 0.000,C 90.000,E1 88.797} C_DIS
LIN {X 0.171,Y -659.830,Z 497.289,A 0.000,B 0.000,C 90.000,E1 88.051} C_DIS
LIN {X -0.010,Y -659.481,Z 497.288,A 0.000,B 0.000,C 90.000,E1 87.822} C_DIS
LIN {X 0.282,Y -658.478,Z 497.285,A 0.000,B 0.000,C 90.000,E1 87.306} C_DIS
LIN {X -0.250,Y -656.557,Z 497.281,A 0.000,B 0.000,C 90.000,E1 86.617} C_DIS
LIN {X 0.015,Y -655.072,Z 497.278,A 0.000,B 0.000,C 90.000,E1 86.102} C_DIS
LIN {X 0.312,Y -653.309,Z 497.276,A 0.000,B 0.000,C 90.000,E1 85.584} C_DIS
LIN {X -0.262,Y -650.271,Z 497.272,A 0.000,B 0.000,C 90.000,E1 84.894} C_DIS
LIN {X -0.105,Y -647.366,Z 497.268,A 0.000,B 0.000,C 90.000,E1 84.261} C_DIS
LIN {X 0.024,Y -644.155,Z 497.265,A 0.000,B 0.000,C 90.000,E1 83.628} C_DIS
LIN {X 0.119,Y -640.644,Z 497.261,A 0.000,B 0.000,C 90.000,E1 82.996} C_DIS
LIN {X 0.264,Y -636.683,Z 497.258,A 0.000,B 0.000,C 90.000,E1 82.356} C_DIS
LIN {X -0.195,Y -633.383,Z 497.255,A 0.000,B 0.000,C 90.000,E1 81.894} C_DIS
LIN {X -0.014,Y -628.961,Z 497.251,A 0.000,B 0.000,C 90.000,E1 81.254} C_DIS
LIN {X -0.113,Y -623.049,Z 497.247,A 0.000,B 0.000,C 90.000,E1 80.500} C_DIS
LIN {X -0.102,Y -617.782,Z 497.244,A 0.000,B 0.000,C 90.000,E1 79.859} C_DIS
LIN {X -0.137,Y -612.084,Z 497.240,A 0.000,B 0.000,C 90.000,E1 79.218} C_DIS
LIN {X -0.108,Y -607.169,Z 497.237,A 0.000,B 0.000,C 90.000,E1 78.701} C_DIS
LIN {X 0.224,Y -600.785,Z 497.234,A 0.000,B 0.000,C 90.000,E1 78.049} C_DIS
LIN {X 0.055,Y -596.756,Z 497.232,A 0.000,B 0.000,C 90.000,E1 77.701} C_DIS
LIN {X 0.136,Y -590.946,Z 497.229,A 0.000,B 0.000,C 90.000,E1 77.229} C_DIS
LIN {X -0.261,Y -582.361,Z 497.226,A 0.000,B 0.000,C 90.000,E1 76.645} C_DIS
LIN {X -0.013,Y -579.221,Z 497.225,A 0.000,B 0.000,C 90.000,E1 76.408} C_DIS
LIN {X 0.292,Y -572.743,Z 497.222,A 0.000,B 0.000,C 90.000,E1 75.992} C_DIS
LIN {X 0.074,Y -567.832,Z 497.221,A 0.000,B 0.000,C 90.000,E1 75.755} C_DIS
LIN {X -0.016,Y -561.012,Z 497.219,A 0.000,B 0.000,C 90.000,E1 75.463} C_DIS
LIN {X 0.140,Y -555.365,Z 497.218,A 0.000,B 0.000,C 90.000,E1 75.227} C_DIS
LIN {X 0.176,Y -549.729,Z 497.217,A 0.000,B 0.000,C 90.000,E1 75.046} C_DIS
LIN {X -0.273,Y -543.414,Z 497.216,A 0.000,B 0.000,C 90.000,E1 74.936} C_DIS
LIN {X -0.203,Y -537.598,Z 497.216,A 0.000,B 0.000,C 90.000,E1 74.810} C_DIS
LIN {X 0.306,Y -529.160,Z 497.215,A 0.000,B 0.000,C 90.000,E1 74.629} C_DIS
LIN {X 0.086,Y -521.878,Z 497.214,A 0.000,B 0.000,C 90.000,E1 74.574} C_DIS
LIN {X -0.088,Y -509.947,Z 497.214,A 0.000,B 0.000,C 90.000,E1 74.519} C_DIS
LIN {X 0.107,Y -499.268,Z 497.214,A 0.000,B 0.000,C 90.000,E1 74.464} C_DIS
LIN {X 0.180,Y -493.421,Z 497.214,A 0.000,B 0.000,C 90.000,E1 74.448} C_DIS
LIN {X 0.145,Y -476.909,Z 497.214,A 0.000,B 0.000,C 90.000,E1 74.448} C_DIS
LIN {X 0.137,Y -473.980,Z 497.200,A 0.000,B 0.000,C 90.000,E1 71.945} C_DIS
LIN {X 0.261,Y -466.345,Z 497.175,A 0.000,B 0.000,C 90.000,E1 67.539} C_DIS
LIN {X 0.146,Y -465.385,Z 497.172,A 0.000,B 0.000,C 90.000,E1 66.922} C_DIS
LIN {X 0.114,Y -456.971,Z 497.149,A 0.000,B 0.000,C 90.000,E1 62.794} C_DIS
LIN {X 0.009,Y -455.369,Z 497.144,A 0.000,B 0.000,C 90.000,E1 61.847} C_DIS
LIN {X -0.124,Y -450.412,Z 497.132,A 0.000,B 0.000,C 90.000,E1 59.793} C_DIS
LIN {X -0.164,Y -450.427,Z 497.132,A 0.000,B 0.000,C 90.000,E1 59.793} C_DIS
LIN {X -0.014,Y -455.159,Z 497.127,A 0.000,B 0.000,C 90.000,E1 58.791} C_DIS
LIN {X -0.079,Y -459.505,Z 497.121,A 0.000,B 0.000,C 90.000,E1 57.837} C_DIS
LIN {X 0.170,Y -461.475,Z 497.119,A 0.000,B 0.000,C 90.000,E1 57.327} C_DIS
LIN {X -0.214,Y -465.112,Z 497.113,A 0.000,B 0.000,C 90.000,E1 56.421} C_DIS
LIN {X -0.178,Y -468.178,Z 497.108,A 0.000,B 0.000,C 90.000,E1 55.468} C_DIS
LIN {X 0.005,Y -469.962,Z 497.105,A 0.000,B 0.000,C 90.000,E1 54.815} C_DIS
LIN {X 0.089,Y -472.135,Z 497.099,A 0.000,B 0.000,C 90.000,E1 53.863} C_DIS
LIN {X -0.071,Y -473.409,Z 497.096,A 0.000,B 0.000,C 90.000,E1 53.256} C_DIS
LIN {X -0.047,Y -474.903,Z 497.091,A 0.000,B 0.000,C 90.000,E1 52.316} C_DIS
LIN {X -0.006,Y -476.249,Z 497.085,A 0.000,B 0.000,C 90.000,E1 51.376} C_DIS
LIN {X 0.045,Y -477.258,Z 497.080,A 0.000,B 0.000,C 90.000,E1 50.436} C_DIS
LIN {X 0.313,Y -478.612,Z 497.072,A 0.000,B 0.000,C 90.000,E1 48.852} C_DIS
LIN {X 0.130,Y -479.391,Z 497.065,A 0.000,B 0.000,C 90.000,E1 47.634} C_DIS
LIN {X 0.160,Y -479.857,Z 497.060,A 0.000,B 0.000,C 90.000,E1 46.701} C_DIS
LIN {X -0.029,Y -480.169,Z 497.053,A 0.000,B 0.000,C 90.000,E1 45.486} C_DIS
LIN {X 0.001,Y -480.329,Z 497.048,A 0.000,B 0.000,C 90.000,E1 44.555} C_DIS
LIN {X 0.160,Y -480.320,Z 497.041,A 0.000,B 0.000,C 90.000,E1 43.299} C_DIS
LIN {X 0.200,Y -480.136,Z 497.036,A 0.000,B 0.000,C 90.000,E1 42.366} C_DIS
LIN {X -0.080,Y -479.820,Z 497.030,A 0.000,B 0.000,C 90.000,E1 41.472} C_DIS
LIN {X -0.133,Y -479.052,Z 497.022,A 0.000,B 0.000,C 90.000,E1 39.930} C_DIS
LIN {X 0.052,Y -478.432,Z 497.015,A 0.000,B 0.000,C 90.000,E1 38.669} C_DIS
LIN {X 0.200,Y -477.369,Z 497.005,A 0.000,B 0.000,C 90.000,E1 36.790} C_DIS
LIN {X -0.219,Y -476.584,Z 496.998,A 0.000,B 0.000,C 90.000,E1 35.598} C_DIS
LIN {X -0.012,Y -475.086,Z 496.987,A 0.000,B 0.000,C 90.000,E1 33.706} C_DIS
LIN {X 0.107,Y -473.795,Z 496.979,A 0.000,B 0.000,C 90.000,E1 32.133} C_DIS
LIN {X 0.176,Y -472.688,Z 496.972,A 0.000,B 0.000,C 90.000,E1 30.875} C_DIS
LIN {X -0.004,Y -471.131,Z 496.963,A 0.000,B 0.000,C 90.000,E1 29.333} C_DIS
LIN {X -0.040,Y -469.597,Z 496.954,A 0.000,B 0.000,C 90.000,E1 27.769} C_DIS
LIN {X -0.229,Y -467.687,Z 496.942,A 0.000,B 0.000,C 90.000,E1 25.591} C_DIS
LIN {X 0.060,Y -465.495,Z 496.926,A 0.000,B 0.000,C 90.000,E1 22.717} C_DIS
LIN {X -0.067,Y -463.826,Z 496.910,A 0.000,B 0.000,C 90.000,E1 19.885} C_DIS
LIN {X -0.204,Y -462.878,Z 496.900,A 0.000,B 0.000,C 90.000,E1 18.000} C_DIS
LIN {X 0.071,Y -461.841,Z 496.886,A 0.000,B 0.000,C 90.000,E1 15.426} C_DIS
LIN {X -0.145,Y -461.085,Z 496.870,A 0.000,B 0.000,C 90.000,E1 12.591} C_DIS
LIN {X -0.139,Y -460.870,Z 496.854,A 0.000,B 0.000,C 90.000,E1 9.726} C_DIS
LIN {X -0.156,Y -461.211,Z 496.840,A 0.000,B 0.000,C 90.000,E1 7.182} C_DIS
LIN {X -0.035,Y -462.495,Z 496.820,A 0.000,B 0.000,C 90.000,E1 3.669} C_DIS
LIN {X -0.157,Y -464.071,Z 496.806,A 0.000,B 0.000,C 90.000,E1 1.146} C_DIS
LIN {X 0.139,Y -466.219,Z 496.792,A 0.000,B 0.000,C 90.000,E1 358.511} C_DIS
LIN {X 0.146,Y -468.246,Z 496.781,A 0.000,B 0.000,C 90.000,E1 356.617} C_DIS
LIN {X -0.226,Y -471.199,Z 496.767,A 0.000,B 0.000,C 90.000,E1 354.147} C_DIS
LIN {X 0.158,Y -473.198,Z 496.759,A 0.000,B 0.000,C 90.000,E1 352.534} C_DIS
LIN {X -0.155,Y -476.113,Z 496.747,A 0.000,B 0.000,C 90.000,E1 350.387} C_DIS
LIN {X 0.018,Y -479.974,Z 496.733,A 0.000,B 0.000,C 90.000,E1 347.881} C_DIS
LIN {X 0.181,Y -483.906,Z 496.721,A 0.000,B 0.000,C 90.000,E1 345.700} C_DIS
LIN {X -0.019,Y -488.901,Z 496.707,A 0.000,B 0.000,C 90.000,E1 343.268} C_DIS
LIN {X -0.177,Y -492.781,Z 496.697,A 0.000,B 0.000,C 90.000,E1 341.456} C_DIS
LIN {X -0.078,Y -496.861,Z 496.687,A 0.000,B 0.000,C 90.000,E1 339.625} C_DIS
LIN {X 0.111,Y -500.840,Z 496.677,A 0.000,B 0.000,C 90.000,E1 337.794} C_DIS
LIN {X -0.059,Y -503.431,Z 496.670,A 0.000,B 0.000,C 90.000,E1 336.613} C_DIS
LIN {X 0.190,Y -507.195,Z 496.660,A 0.000,B 0.000,C 90.000,E1 334.793} C_DIS
LIN {X -0.073,Y -511.500,Z 496.649,A 0.000,B 0.000,C 90.000,E1 332.743} C_DIS
LIN {X 0.023,Y -517.135,Z 496.634,A 0.000,B 0.000,C 90.000,E1 330.078} C_DIS
LIN {X -0.019,Y -522.319,Z 496.621,A 0.000,B 0.000,C 90.000,E1 327.740} C_DIS
LIN {X 0.220,Y -527.600,Z 496.608,A 0.000,B 0.000,C 90.000,E1 325.388} C_DIS
LIN {X -0.206,Y -530.951,Z 496.600,A 0.000,B 0.000,C 90.000,E1 323.989} C_DIS
LIN {X -0.267,Y -535.022,Z 496.590,A 0.000,B 0.000,C 90.000,E1 322.271} C_DIS
LIN {X 0.087,Y -538.968,Z 496.581,A 0.000,B 0.000,C 90.000,E1 320.517} C_DIS
LIN {X -0.302,Y -542.945,Z 496.571,A 0.000,B 0.000,C 90.000,E1 318.852} C_DIS
LIN {X 0.130,Y -546.227,Z 496.563,A 0.000,B 0.000,C 90.000,E1 317.391} C_DIS
LIN {X 0.223,Y -549.380,Z 496.556,A 0.000,B 0.000,C 90.000,E1 315.972} C_DIS
LIN {X 0.007,Y -553.019,Z 496.546,A 0.000,B 0.000,C 90.000,E1 314.312} C_DIS
LIN {X -0.163,Y -556.051,Z 496.538,A 0.000,B 0.000,C 90.000,E1 312.933} C_DIS
LIN {X -0.343,Y -558.478,Z 496.532,A 0.000,B 0.000,C 90.000,E1 311.838} C_DIS
LIN {X 0.017,Y -561.510,Z 496.525,A 0.000,B 0.000,C 90.000,E1 310.415} C_DIS
LIN {X 0.105,Y -565.046,Z 496.515,A 0.000,B 0.000,C 90.000,E1 308.749} C_DIS
LIN {X -0.202,Y -569.848,Z 496.503,A 0.000,B 0.000,C 90.000,E1 306.583} C_DIS
LIN {X 0.264,Y -573.541,Z 496.494,A 0.000,B 0.000,C 90.000,E1 304.898} C_DIS
LIN {X 0.008,Y -577.244,Z 496.485,A 0.000,B 0.000,C 90.000,E1 303.293} C_DIS
LIN {X -0.008,Y -580.907,Z 496.476,A 0.000,B 0.000,C 90.000,E1 301.671} C_DIS
LIN {X -0.114,Y -583.689,Z 496.469,A 0.000,B 0.000,C 90.000,E1 300.335} C_DIS
LIN {X -0.054,Y -585.814,Z 496.463,A 0.000,B 0.000,C 90.000,E1 299.255} C_DIS
LIN {X 0.139,Y -588.244,Z 496.455,A 0.000,B 0.000,C 90.000,E1 297.897} C_DIS
LIN {X -0.306,Y -589.902,Z 496.449,A 0.000,B 0.000,C 90.000,E1 296.873} C_DIS
LIN {X -0.093,Y -590.980,Z 496.445,A 0.000,B 0.000,C 90.000,E1 296.052} C_DIS
LIN {X 0.037,Y -592.303,Z 496.439,A 0.000,B 0.000,C 90.000,E1 294.975} C_DIS
LIN {X 0.184,Y -593.319,Z 496.433,A 0.000,B 0.000,C 90.000,E1 293.898} C_DIS
LIN {X 0.008,Y -594.350,Z 496.426,A 0.000,B 0.000,C 90.000,E1 292.589} C_DIS
LIN {X 0.296,Y -595.461,Z 496.417,A 0.000,B 0.000,C 90.000,E1 290.972} C_DIS
LIN {X -0.079,Y -596.196,Z 496.409,A 0.000,B 0.000,C 90.000,E1 289.685} C_DIS
LIN {X -0.188,Y -596.746,Z 496.401,A 0.000,B 0.000,C 90.000,E1 288.109} C_DIS
LIN {X -0.351,Y -597.212,Z 496.393,A 0.000,B 0.000,C 90.000,E1 286.804} C_DIS
LIN {X -0.043,Y -597.650,Z 496.384,A 0.000,B 0.000,C 90.000,E1 285.190} C_DIS
LIN {X 0.108,Y -597.895,Z 496.379,A 0.000,B 0.000,C 90.000,E1 284.120} C_DIS
LIN {X 0.124,Y -598.110,Z 496.370,A 0.000,B 0.000,C 90.000,E1 282.535} C_DIS
LIN {X -0.152,Y -598.180,Z 496.362,A 0.000,B 0.000,C 90.000,E1 281.243} C_DIS
LIN {X 0.043,Y -598.132,Z 496.355,A 0.000,B 0.000,C 90.000,E1 279.905} C_DIS
LIN {X 0.237,Y -597.923,Z 496.348,A 0.000,B 0.000,C 90.000,E1 278.568} C_DIS
LIN {X -0.257,Y -597.556,Z 496.340,A 0.000,B 0.000,C 90.000,E1 277.296} C_DIS
LIN {X 0.147,Y -597.154,Z 496.335,A 0.000,B 0.000,C 90.000,E1 276.201} C_DIS
LIN {X 0.170,Y -596.376,Z 496.327,A 0.000,B 0.000,C 90.000,E1 274.878} C_DIS
LIN {X -0.042,Y -595.610,Z 496.321,A 0.000,B 0.000,C 90.000,E1 273.841} C_DIS
LIN {X 0.283,Y -594.725,Z 496.315,A 0.000,B 0.000,C 90.000,E1 272.751} C_DIS
LIN {X 0.000,Y -593.604,Z 496.310,A 0.000,B 0.000,C 90.000,E1 271.718} C_DIS
LIN {X 0.277,Y -592.328,Z 496.304,A 0.000,B 0.000,C 90.000,E1 270.630} C_DIS
LIN {X 0.158,Y -590.576,Z 496.296,A 0.000,B 0.000,C 90.000,E1 269.312} C_DIS
LIN {X 0.225,Y -588.304,Z 496.287,A 0.000,B 0.000,C 90.000,E1 267.707} C_DIS
LIN {X -0.137,Y -586.736,Z 496.281,A 0.000,B 0.000,C 90.000,E1 266.674} C_DIS
LIN {X 0.243,Y -584.711,Z 496.274,A 0.000,B 0.000,C 90.000,E1 265.298} C_DIS
